LIN {X 0,Y 319.596,Z 143.485,A -85,B 0,C 180,E1 -15098.048,E2 -15098.048} C_VEL
LIN {X 0,Y 319.687,Z 143.47,A -85,B 0,C 180,E1 -15100.962,E2 -15100.962} C_VEL
LIN {X 0,Y 319.73,Z 143.468,A -85,B 0,C 180,E1 -15105.276,E2 -15105.276} C_VEL
LIN {X 0,Y 319.758,Z 143.463,A -85,B 0,C 180,E1 -15109.873,E2 -15109.873} C_VEL
LIN {X 0,Y 319.932,Z 143.443,A -85,B 0,C 180,E1 -15112.426,E2 -15112.426} C_VEL
LIN {X 0,Y 319.746,Z 143.466,A -85,B 0,C 180,E1 -15114.956,E2 -15114.956} C_VEL
LIN {X 0,Y 319.99,Z 143.436,A -85,B 0,C 180,E1 -15117.482,E2 -15117.482} C_VEL
LIN {X 0,Y 320.149,Z 143.413,A -85,B 0,C 180,E1 -15120,E2 -15120} C_VEL
LIN {X 0,Y 319.989,Z 143.434,A -85,B 0,C 180,E1 -15122.517,E2 -15122.517} C_VEL
LIN {X 0,Y 319.953,Z 143.441,A -85,B 0,C 180,E1 -15126.305,E2 -15126.305} C_VEL
LIN {X 0,Y 319.841,Z 143.451,A -85,B 0,C 180,E1 -15128.848,E2 -15128.848} C_VEL
LIN {X 0,Y 319.68,Z 143.472,A -85,B 0,C 180,E1 -15132.7,E2 -15132.7} C_VEL
LIN {X 0,Y 319.698,Z 143.476,A -85,B 0,C 180,E1 -15135.295,E2 -15135.295} C_VEL
LIN {X 0,Y 319.673,Z 143.474,A -85,B 0,C 180,E1 -15139.255,E2 -15139.255} C_VEL
LIN {X 0,Y 319.568,Z 143.491,A -85,B 0,C 180,E1 -15143.319,E2 -15143.319} C_VEL
LIN {X 0,Y 319.633,Z 143.478,A -85,B 0,C 180,E1 -15146.088,E2 -15146.088} C_VEL
LIN {X 0,Y 319.588,Z 143.487,A -85,B 0,C 180,E1 -15148.934,E2 -15148.934} C_VEL
LIN {X 0,Y 319.53,Z 143.493,A -85,B 0,C 180,E1 -15151.862,E2 -15151.862} C_VEL
LIN {X 0,Y 319.577,Z 143.485,A -85,B 0,C 180,E1 -15155.543,E2 -15155.543} C_VEL
LIN {X 0,Y 319.555,Z 143.491,A -85,B 0,C 180,E1 -15158.01,E2 -15158.01} C_VEL
LIN {X 0,Y 319.523,Z 143.488,A -85,B 0,C 180,E1 -15161.597,E2 -15161.597} C_VEL
LIN {X 0,Y 319.486,Z 143.494,A -85,B 0,C 180,E1 -15165.257,E2 -15165.257} C_VEL
LIN {X 0,Y 319.526,Z 143.494,A -85,B 0,C 180,E1 -15168.712,E2 -15168.712} C_VEL
LIN {X 0,Y 319.553,Z 143.489,A -85,B 0,C 180,E1 -15172.35,E2 -15172.35} C_VEL
LIN {X 0,Y 319.559,Z 143.49,A -85,B 0,C 180,E1 -15175.124,E2 -15175.124} C_VEL
LIN {X 0,Y 319.569,Z 143.49,A -85,B 0,C 180,E1 -15179.058,E2 -15179.058} C_VEL
LIN {X 0,Y 319.702,Z 143.582,A -85,B 0,C 180,E1 -15182.596,E2 -15182.596} C_VEL
LIN {X 0,Y 321.213,Z 151.646,A -85,B 0,C 180,E1 -15185.436,E2 -15185.436} C_VEL
LIN {X 0,Y 321.936,Z 156.902,A -85,B 0,C 180,E1 -15187.202,E2 -15187.202} C_VEL
LIN {X 0,Y 320.97,Z 166.795,A -85,B 0,C 180,E1 -15190.25,E2 -15190.25} C_VEL
LIN {X 0,Y 321.774,Z 171.894,A -85,B 0,C 180,E1 -15190.48,E2 -15190.48} C_VEL
LIN {X 0,Y 325.641,Z 196.853,A -85,B 0,C 180,E1 -15191.289,E2 -15191.289} C_VEL
LIN {X 0,Y 325.841,Z 203.062,A -85,B 0,C 180,E1 -15191.442,E2 -15191.442} C_VEL
LIN {X 0,Y 325.186,Z 243.218,A -85,B 0,C 180,E1 -15192.351,E2 -15192.351} C_VEL
LIN {X 0,Y 324.747,Z 252.267,A -85,B 0,C 180,E1 -15192.689,E2 -15192.689} C_VEL
LIN {X 0,Y 324.141,Z 261.891,A -85,B 0,C 180,E1 -15193.224,E2 -15193.224} C_VEL
LIN {X 0,Y 323.392,Z 271.027,A -85,B 0,C 180,E1 -15193.914,E2 -15193.914} C_VEL
LIN {X 0,Y 322.429,Z 281.805,A -85,B 0,C 180,E1 -15194.999,E2 -15194.999} C_VEL
LIN {X 0,Y 321.43,Z 290.08,A -85,B 0,C 180,E1 -15196.084,E2 -15196.084} C_VEL
LIN {X 0,Y 320.528,Z 297.765,A -85,B 0,C 180,E1 -15197.335,E2 -15197.335} C_VEL
LIN {X 0,Y 319.789,Z 304.092,A -85,B 0,C 180,E1 -15198.592,E2 -15198.592} C_VEL
LIN {X 0,Y 319.189,Z 309.35,A -85,B 0,C 180,E1 -15199.855,E2 -15199.855} C_VEL
LIN {X 0,Y 318.696,Z 313.734,A -85,B 0,C 180,E1 -15201.12,E2 -15201.12} C_VEL
LIN {X 0,Y 318.206,Z 318.906,A -85,B 0,C 180,E1 -15203.023,E2 -15203.023} C_VEL
LIN {X 0,Y 317.889,Z 322.703,A -85,B 0,C 180,E1 -15204.927,E2 -15204.927} C_VEL
LIN {X 0,Y 317.831,Z 324.448,A -85,B 0,C 180,E1 -15206.197,E2 -15206.197} C_VEL
LIN {X 0,Y 317.746,Z 325.696,A -85,B 0,C 180,E1 -15207.465,E2 -15207.465} C_VEL
LIN {X 0,Y 317.695,Z 326.471,A -85,B 0,C 180,E1 -15208.733,E2 -15208.733} C_VEL
LIN {X 0,Y 317.717,Z 326.765,A -85,B 0,C 180,E1 -15210,E2 -15210} C_VEL
LIN {X 0,Y 317.695,Z 326.466,A -85,B 0,C 180,E1 -15211.268,E2 -15211.268} C_VEL
LIN {X 0,Y 317.746,Z 325.679,A -85,B 0,C 180,E1 -15212.536,E2 -15212.536} C_VEL
LIN {X 0,Y 317.831,Z 324.419,A -85,B 0,C 180,E1 -15213.804,E2 -15213.804} C_VEL
LIN {X 0,Y 317.886,Z 322.663,A -85,B 0,C 180,E1 -15215.074,E2 -15215.074} C_VEL
LIN {X 0,Y 318.204,Z 318.854,A -85,B 0,C 180,E1 -15216.978,E2 -15216.978} C_VEL
LIN {X 0,Y 318.625,Z 313.665,A -85,B 0,C 180,E1 -15218.882,E2 -15218.882} C_VEL
LIN {X 0,Y 319.453,Z 306.829,A -85,B 0,C 180,E1 -15220.778,E2 -15220.778} C_VEL
LIN {X 0,Y 320.323,Z 299.357,A -85,B 0,C 180,E1 -15222.352,E2 -15222.352} C_VEL
LIN {X 0,Y 321.234,Z 291.99,A -85,B 0,C 180,E1 -15223.603,E2 -15223.603} C_VEL
LIN {X 0,Y 322.109,Z 284.099,A -85,B 0,C 180,E1 -15224.693,E2 -15224.693} C_VEL
LIN {X 0,Y 322.956,Z 275.758,A -85,B 0,C 180,E1 -15225.623,E2 -15225.623} C_VEL
LIN {X 0,Y 323.876,Z 265.096,A -85,B 0,C 180,E1 -15226.548,E2 -15226.548} C_VEL
LIN {X 0,Y 324.637,Z 253.466,A -85,B 0,C 180,E1 -15227.237,E2 -15227.237} C_VEL
LIN {X 0,Y 325.161,Z 243.694,A -85,B 0,C 180,E1 -15227.614,E2 -15227.614} C_VEL
LIN {X 0,Y 325.684,Z 197.491,A -85,B 0,C 180,E1 -15228.671,E2 -15228.671} C_VEL
LIN {X 0,Y 322.039,Z 173.379,A -85,B 0,C 180,E1 -15229.446,E2 -15229.446} C_VEL
LIN {X 0,Y 320.97,Z 166.868,A -85,B 0,C 180,E1 -15229.716,E2 -15229.716} C_VEL
LIN {X 0,Y 321.896,Z 157.872,A -85,B 0,C 180,E1 -15232.463,E2 -15232.463} C_VEL
LIN {X 0,Y 321.503,Z 153.471,A -85,B 0,C 180,E1 -15233.919,E2 -15233.919} C_VEL
LIN {X 0,Y 319.722,Z 143.707,A -85,B 0,C 180,E1 -15237.314,E2 -15237.314} C_VEL
LIN {X 0,Y 319.59,Z 143.475,A -85,B 0,C 180,E1 -15238.934,E2 -15238.934} C_VEL
LIN {X 0,Y 319.533,Z 143.496,A -85,B 0,C 180,E1 -15241.862,E2 -15241.862} C_VEL
LIN {X 0,Y 319.58,Z 143.488,A -85,B 0,C 180,E1 -15245.543,E2 -15245.543} C_VEL
LIN {X 0,Y 319.557,Z 143.486,A -85,B 0,C 180,E1 -15248.01,E2 -15248.01} C_VEL
LIN {X 0,Y 319.526,Z 143.496,A -85,B 0,C 180,E1 -15251.597,E2 -15251.597} C_VEL
LIN {X 0,Y 319.488,Z 143.494,A -85,B 0,C 180,E1 -15255.257,E2 -15255.257} C_VEL
LIN {X 0,Y 319.528,Z 143.488,A -85,B 0,C 180,E1 -15258.712,E2 -15258.712} C_VEL
LIN {X 0,Y 319.562,Z 143.489,A -85,B 0,C 180,E1 -15262.348,E2 -15262.348} C_VEL
LIN {X 0,Y 319.561,Z 143.489,A -85,B 0,C 180,E1 -15265.124,E2 -15265.124} C_VEL
LIN {X 0,Y 319.571,Z 143.492,A -85,B 0,C 180,E1 -15269.058,E2 -15269.058} C_VEL
LIN {X 0,Y 319.609,Z 143.479,A -85,B 0,C 180,E1 -15272.498,E2 -15272.498} C_VEL
LIN {X 0,Y 319.606,Z 143.486,A -85,B 0,C 180,E1 -15275.304,E2 -15275.304} C_VEL
LIN {X 0,Y 319.599,Z 143.483,A -85,B 0,C 180,E1 -15278.048,E2 -15278.048} C_VEL
LIN {X 0,Y 319.69,Z 143.472,A -85,B 0,C 180,E1 -15280.962,E2 -15280.962} C_VEL
LIN {X 0,Y 319.732,Z 143.468,A -85,B 0,C 180,E1 -15285.276,E2 -15285.276} C_VEL
LIN {X 0,Y 319.754,Z 143.458,A -85,B 0,C 180,E1 -15289.873,E2 -15289.873} C_VEL
LIN {X 0,Y 319.914,Z 143.449,A -85,B 0,C 180,E1 -15292.426,E2 -15292.426} C_VEL
LIN {X 0,Y 319.746,Z 143.466,A -85,B 0,C 180,E1 -15294.956,E2 -15294.956} C_VEL
LIN {X 0,Y 319.991,Z 143.433,A -85,B 0,C 180,E1 -15297.483,E2 -15297.483} C_VEL
LIN {X 0,Y 320.133,Z 143.415,A -85,B 0,C 180,E1 -15300,E2 -15300} C_VEL
LIN {X 0,Y 319.991,Z 143.436,A -85,B 0,C 180,E1 -15302.518,E2 -15302.518} C_VEL
LIN {X 0,Y 319.934,Z 143.44,A -85,B 0,C 180,E1 -15306.638,E2 -15306.638} C_VEL
LIN {X 0,Y 319.762,Z 143.463,A -85,B 0,C 180,E1 -15310.127,E2 -15310.127} C_VEL
LIN {X 0,Y 319.733,Z 143.467,A -85,B 0,C 180,E1 -15314.724,E2 -15314.724} C_VEL
LIN {X 0,Y 319.691,Z 143.469,A -85,B 0,C 180,E1 -15319.038,E2 -15319.038} C_VEL
LIN {X 0,Y 319.572,Z 143.491,A -85,B 0,C 180,E1 -15323.319,E2 -15323.319} C_VEL
LIN {X 0,Y 319.62,Z 143.477,A -85,B 0,C 180,E1 -15326.089,E2 -15326.089} C_VEL
LIN {X 0,Y 319.591,Z 143.488,A -85,B 0,C 180,E1 -15328.934,E2 -15328.934} C_VEL
LIN {X 0,Y 319.534,Z 143.492,A -85,B 0,C 180,E1 -15331.862,E2 -15331.862} C_VEL
LIN {X 0,Y 319.581,Z 143.486,A -85,B 0,C 180,E1 -15335.543,E2 -15335.543} C_VEL
LIN {X 0,Y 319.559,Z 143.49,A -85,B 0,C 180,E1 -15338.01,E2 -15338.01} C_VEL
LIN {X 0,Y 319.527,Z 143.493,A -85,B 0,C 180,E1 -15341.597,E2 -15341.597} C_VEL
LIN {X 0,Y 319.49,Z 143.495,A -85,B 0,C 180,E1 -15345.257,E2 -15345.257} C_VEL
LIN {X 0,Y 319.53,Z 143.49,A -85,B 0,C 180,E1 -15348.712,E2 -15348.712} C_VEL
LIN {X 0,Y 319.579,Z 143.489,A -85,B 0,C 180,E1 -15352.344,E2 -15352.344} C_VEL
LIN {X 0,Y 319.562,Z 143.48,A -85,B 0,C 180,E1 -15355.123,E2 -15355.123} C_VEL
LIN {X 0,Y 319.572,Z 143.488,A -85,B 0,C 180,E1 -15359.058,E2 -15359.058} C_VEL
LIN {X 0,Y 319.61,Z 143.483,A -85,B 0,C 180,E1 -15362.498,E2 -15362.498} C_VEL
LIN {X 0,Y 319.635,Z 143.653,A -85,B 0,C 180,E1 -15365.955,E2 -15365.955} C_VEL
LIN {X 0,Y 321.074,Z 151.506,A -85,B 0,C 180,E1 -15368.828,E2 -15368.828} C_VEL
LIN {X 0,Y 321.228,Z 156.146,A -85,B 0,C 180,E1 -15370.342,E2 -15370.342} C_VEL
LIN {X 0,Y 321.834,Z 159.261,A -85,B 0,C 180,E1 -15370.514,E2 -15370.514} C_VEL
LIN {X 0,Y 326.078,Z 182.285,A -85,B 0,C 180,E1 -15371.305,E2 -15371.305} C_VEL
LIN {X 0,Y 325.231,Z 232.335,A -85,B 0,C 180,E1 -15372.431,E2 -15372.431} C_VEL
LIN {X 0,Y 324.852,Z 242.15,A -85,B 0,C 180,E1 -15372.815,E2 -15372.815} C_VEL
LIN {X 0,Y 324.282,Z 253.252,A -85,B 0,C 180,E1 -15373.474,E2 -15373.474} C_VEL
LIN {X 0,Y 323.393,Z 264.079,A -85,B 0,C 180,E1 -15374.399,E2 -15374.399} C_VEL
LIN {X 0,Y 322.546,Z 272.474,A -85,B 0,C 180,E1 -15375.327,E2 -15375.327} C_VEL
LIN {X 0,Y 321.773,Z 280.397,A -85,B 0,C 180,E1 -15376.42,E2 -15376.42} C_VEL
LIN {X 0,Y 321.069,Z 286.089,A -85,B 0,C 180,E1 -15377.356,E2 -15377.356} C_VEL
LIN {X 0,Y 320.328,Z 292.441,A -85,B 0,C 180,E1 -15378.611,E2 -15378.611} C_VEL
LIN {X 0,Y 319.592,Z 297.723,A -85,B 0,C 180,E1 -15379.867,E2 -15379.867} C_VEL
LIN {X 0,Y 319.125,Z 302.13,A -85,B 0,C 180,E1 -15381.132,E2 -15381.132} C_VEL
LIN {X 0,Y 318.731,Z 305.8,A -85,B 0,C 180,E1 -15382.397,E2 -15382.397} C_VEL
LIN {X 0,Y 318.383,Z 308.798,A -85,B 0,C 180,E1 -15383.663,E2 -15383.663} C_VEL
LIN {X 0,Y 318.189,Z 311.118,A -85,B 0,C 180,E1 -15384.931,E2 -15384.931} C_VEL
LIN {X 0,Y 317.988,Z 312.884,A -85,B 0,C 180,E1 -15386.198,E2 -15386.198} C_VEL
LIN {X 0,Y 317.81,Z 314.158,A -85,B 0,C 180,E1 -15387.465,E2 -15387.465} C_VEL
LIN {X 0,Y 317.725,Z 314.961,A -85,B 0,C 180,E1 -15388.732,E2 -15388.732} C_VEL
LIN {X 0,Y 317.721,Z 315.267,A -85,B 0,C 180,E1 -15390,E2 -15390} C_VEL
LIN {X 0,Y 317.725,Z 314.99,A -85,B 0,C 180,E1 -15391.267,E2 -15391.267} C_VEL
LIN {X 0,Y 317.808,Z 314.243,A -85,B 0,C 180,E1 -15392.535,E2 -15392.535} C_VEL
LIN {X 0,Y 317.984,Z 313.027,A -85,B 0,C 180,E1 -15393.801,E2 -15393.801} C_VEL
LIN {X 0,Y 318.265,Z 310.175,A -85,B 0,C 180,E1 -15395.703,E2 -15395.703} C_VEL
LIN {X 0,Y 318.578,Z 307.161,A -85,B 0,C 180,E1 -15397.144,E2 -15397.144} C_VEL
LIN {X 0,Y 319.063,Z 302.468,A -85,B 0,C 180,E1 -15398.869,E2 -15398.869} C_VEL
LIN {X 0,Y 319.729,Z 296.969,A -85,B 0,C 180,E1 -15400.448,E2 -15400.448} C_VEL
LIN {X 0,Y 320.595,Z 290.059,A -85,B 0,C 180,E1 -15402.02,E2 -15402.02} C_VEL
LIN {X 0,Y 321.555,Z 282.123,A -85,B 0,C 180,E1 -15403.428,E2 -15403.428} C_VEL
LIN {X 0,Y 322.403,Z 274.555,A -85,B 0,C 180,E1 -15404.518,E2 -15404.518} C_VEL
LIN {X 0,Y 323.255,Z 266.621,A -85,B 0,C 180,E1 -15405.446,E2 -15405.446} C_VEL
LIN {X 0,Y 323.921,Z 258.426,A -85,B 0,C 180,E1 -15406.221,E2 -15406.221} C_VEL
LIN {X 0,Y 324.56,Z 250.118,A -85,B 0,C 180,E1 -15406.835,E2 -15406.835} C_VEL
LIN {X 0,Y 325.022,Z 241.136,A -85,B 0,C 180,E1 -15407.337,E2 -15407.337} C_VEL
LIN {X 0,Y 325.384,Z 231.483,A -85,B 0,C 180,E1 -15407.7,E2 -15407.7} C_VEL
LIN {X 0,Y 326.088,Z 182.324,A -85,B 0,C 180,E1 -15408.806,E2 -15408.806} C_VEL
LIN {X 0,Y 321.573,Z 158.002,A -85,B 0,C 180,E1 -15409.646,E2 -15409.646} C_VEL
LIN {X 0,Y 321.227,Z 156.132,A -85,B 0,C 180,E1 -15409.774,E2 -15409.774} C_VEL
LIN {X 0,Y 321.084,Z 151.844,A -85,B 0,C 180,E1 -15411.171,E2 -15411.171} C_VEL
LIN {X 0,Y 319.679,Z 143.603,A -85,B 0,C 180,E1 -15414.192,E2 -15414.192} C_VEL
LIN {X 0,Y 319.609,Z 143.482,A -85,B 0,C 180,E1 -15417.501,E2 -15417.501} C_VEL
LIN {X 0,Y 319.57,Z 143.488,A -85,B 0,C 180,E1 -15420.942,E2 -15420.942} C_VEL
LIN {X 0,Y 319.56,Z 143.481,A -85,B 0,C 180,E1 -15424.876,E2 -15424.876} C_VEL
LIN {X 0,Y 319.57,Z 143.492,A -85,B 0,C 180,E1 -15428.037,E2 -15428.037} C_VEL
LIN {X 0,Y 319.525,Z 143.489,A -85,B 0,C 180,E1 -15431.597,E2 -15431.597} C_VEL
LIN {X 0,Y 319.515,Z 143.485,A -85,B 0,C 180,E1 -15433.527,E2 -15433.527} C_VEL
LIN {X 0,Y 318.79,Z 143.583,A -85,B 0,C 180,E1 -15434.578,E2 -15434.578} C_VEL
LIN {X 0,Y 315.91,Z 143.945,A -85,B 0,C 180,E1 -15436.289,E2 -15436.289} C_VEL
LIN {X 0,Y 313.527,Z 144.245,A -85,B 0,C 180,E1 -15437.676,E2 -15437.676} C_VEL
LIN {X 0,Y 312.541,Z 144.364,A -85,B 0,C 180,E1 -15438.75,E2 -15438.75} C_VEL
LIN {X 0,Y 312.478,Z 144.373,A -85,B 0,C 180,E1 -15439.113,E2 -15439.113} C_VEL
LIN {X 0,Y 312.524,Z 144.366,A -85,B 0,C 180,E1 -15442.615,E2 -15442.615} C_VEL
LIN {X 0,Y 312.518,Z 144.361,A -85,B 0,C 180,E1 -15446.311,E2 -15446.311} C_VEL
LIN {X 0,Y 312.544,Z 144.363,A -85,B 0,C 180,E1 -15450.35,E2 -15450.35} C_VEL
LIN {X 0,Y 312.596,Z 144.351,A -85,B 0,C 180,E1 -15454.066,E2 -15454.066} C_VEL
LIN {X 0,Y 312.586,Z 144.358,A -85,B 0,C 180,E1 -15457.529,E2 -15457.529} C_VEL
LIN {X 0,Y 312.637,Z 144.344,A -85,B 0,C 180,E1 -15461.656,E2 -15461.656} C_VEL
LIN {X 0,Y 312.693,Z 144.344,A -85,B 0,C 180,E1 -15465.686,E2 -15465.686} C_VEL
LIN {X 0,Y 312.703,Z 144.34,A -85,B 0,C 180,E1 -15469.642,E2 -15469.642} C_VEL
LIN {X 0,Y 312.87,Z 144.32,A -85,B 0,C 180,E1 -15472.254,E2 -15472.254} C_VEL
LIN {X 0,Y 312.716,Z 144.342,A -85,B 0,C 180,E1 -15474.842,E2 -15474.842} C_VEL
LIN {X 0,Y 312.989,Z 144.304,A -85,B 0,C 180,E1 -15478.713,E2 -15478.713} C_VEL
LIN {X 0,Y 312.989,Z 144.3,A -85,B 0,C 180,E1 -15481.287,E2 -15481.287} C_VEL
LIN {X 0,Y 312.718,Z 144.342,A -85,B 0,C 180,E1 -15485.157,E2 -15485.157} C_VEL
LIN {X 0,Y 312.871,Z 144.324,A -85,B 0,C 180,E1 -15487.746,E2 -15487.746} C_VEL
LIN {X 0,Y 312.667,Z 144.347,A -85,B 0,C 180,E1 -15491.671,E2 -15491.671} C_VEL
LIN {X 0,Y 312.698,Z 144.345,A -85,B 0,C 180,E1 -15494.888,E2 -15494.888} C_VEL
LIN {X 0,Y 312.628,Z 144.35,A -85,B 0,C 180,E1 -15499.236,E2 -15499.236} C_VEL
LIN {X 0,Y 312.544,Z 144.365,A -85,B 0,C 180,E1 -15502.789,E2 -15502.789} C_VEL
LIN {X 0,Y 312.581,Z 144.359,A -85,B 0,C 180,E1 -15506.723,E2 -15506.723} C_VEL
LIN {X 0,Y 312.543,Z 144.362,A -85,B 0,C 180,E1 -15509.65,E2 -15509.65} C_VEL
LIN {X 0,Y 312.517,Z 144.364,A -85,B 0,C 180,E1 -15513.689,E2 -15513.689} C_VEL
LIN {X 0,Y 312.523,Z 144.366,A -85,B 0,C 180,E1 -15517.385,E2 -15517.385} C_VEL
LIN {X 0,Y 312.488,Z 144.367,A -85,B 0,C 180,E1 -15520.709,E2 -15520.709} C_VEL
LIN {X 0,Y 312.449,Z 144.363,A -85,B 0,C 180,E1 -15524.21,E2 -15524.21} C_VEL
LIN {X 0,Y 312.482,Z 144.374,A -85,B 0,C 180,E1 -15527.919,E2 -15527.919} C_VEL
LIN {X 0,Y 312.497,Z 144.363,A -85,B 0,C 180,E1 -15530.971,E2 -15530.971} C_VEL
LIN {X 0,Y 312.53,Z 144.368,A -85,B 0,C 180,E1 -15534.221,E2 -15534.221} C_VEL
LIN {X 0,Y 312.504,Z 144.365,A -85,B 0,C 180,E1 -15537.334,E2 -15537.334} C_VEL
LIN {X 0,Y 312.55,Z 144.344,A -85,B 0,C 180,E1 -15541.277,E2 -15541.277} C_VEL
LIN {X 0,Y 312.634,Z 144.484,A -85,B 0,C 180,E1 -15542.287,E2 -15542.287} C_VEL
LIN {X 0,Y 314.194,Z 152.563,A -85,B 0,C 180,E1 -15545.204,E2 -15545.204} C_VEL
LIN {X 0,Y 314.96,Z 157.818,A -85,B 0,C 180,E1 -15547.015,E2 -15547.015} C_VEL
LIN {X 0,Y 314.083,Z 166.45,A -85,B 0,C 180,E1 -15549.756,E2 -15549.756} C_VEL
LIN {X 0,Y 314.392,Z 168.734,A -85,B 0,C 180,E1 -15549.93,E2 -15549.93} C_VEL
LIN {X 0,Y 318.64,Z 195.359,A -85,B 0,C 180,E1 -15550.83,E2 -15550.83} C_VEL
LIN {X 0,Y 319.138,Z 202.091,A -85,B 0,C 180,E1 -15551.018,E2 -15551.018} C_VEL
LIN {X 0,Y 318.413,Z 243.216,A -85,B 0,C 180,E1 -15551.966,E2 -15551.966} C_VEL
LIN {X 0,Y 317.919,Z 252.979,A -85,B 0,C 180,E1 -15552.346,E2 -15552.346} C_VEL
LIN {X 0,Y 317.288,Z 262.98,A -85,B 0,C 180,E1 -15552.933,E2 -15552.933} C_VEL
LIN {X 0,Y 316.28,Z 274.341,A -85,B 0,C 180,E1 -15553.874,E2 -15553.874} C_VEL
LIN {X 0,Y 315.41,Z 282.912,A -85,B 0,C 180,E1 -15554.823,E2 -15554.823} C_VEL
LIN {X 0,Y 314.397,Z 290.976,A -85,B 0,C 180,E1 -15555.931,E2 -15555.931} C_VEL
LIN {X 0,Y 313.588,Z 297.639,A -85,B 0,C 180,E1 -15557.049,E2 -15557.049} C_VEL
LIN {X 0,Y 312.824,Z 303.966,A -85,B 0,C 180,E1 -15558.335,E2 -15558.335} C_VEL
LIN {X 0,Y 312.197,Z 309.223,A -85,B 0,C 180,E1 -15559.625,E2 -15559.625} C_VEL
LIN {X 0,Y 311.661,Z 313.607,A -85,B 0,C 180,E1 -15560.918,E2 -15560.918} C_VEL
LIN {X 0,Y 311.133,Z 318.778,A -85,B 0,C 180,E1 -15562.864,E2 -15562.864} C_VEL
LIN {X 0,Y 310.807,Z 322.575,A -85,B 0,C 180,E1 -15564.811,E2 -15564.811} C_VEL
LIN {X 0,Y 310.745,Z 324.32,A -85,B 0,C 180,E1 -15566.11,E2 -15566.11} C_VEL
LIN {X 0,Y 310.672,Z 325.568,A -85,B 0,C 180,E1 -15567.407,E2 -15567.407} C_VEL
LIN {X 0,Y 310.612,Z 326.343,A -85,B 0,C 180,E1 -15568.704,E2 -15568.704} C_VEL
LIN {X 0,Y 310.629,Z 326.637,A -85,B 0,C 180,E1 -15570,E2 -15570} C_VEL
LIN {X 0,Y 310.612,Z 326.338,A -85,B 0,C 180,E1 -15571.297,E2 -15571.297} C_VEL
LIN {X 0,Y 310.672,Z 325.551,A -85,B 0,C 180,E1 -15572.593,E2 -15572.593} C_VEL
LIN {X 0,Y 310.745,Z 324.29,A -85,B 0,C 180,E1 -15573.891,E2 -15573.891} C_VEL
LIN {X 0,Y 310.889,Z 321.236,A -85,B 0,C 180,E1 -15575.919,E2 -15575.919} C_VEL
LIN {X 0,Y 311.258,Z 317.201,A -85,B 0,C 180,E1 -15577.786,E2 -15577.786} C_VEL
LIN {X 0,Y 311.899,Z 311.486,A -85,B 0,C 180,E1 -15579.73,E2 -15579.73} C_VEL
LIN {X 0,Y 312.638,Z 305.282,A -85,B 0,C 180,E1 -15581.344,E2 -15581.344} C_VEL
LIN {X 0,Y 313.374,Z 299.226,A -85,B 0,C 180,E1 -15582.631,E2 -15582.631} C_VEL
LIN {X 0,Y 314.34,Z 291.859,A -85,B 0,C 180,E1 -15583.907,E2 -15583.907} C_VEL
LIN {X 0,Y 315.239,Z 283.967,A -85,B 0,C 180,E1 -15585.021,E2 -15585.021} C_VEL
LIN {X 0,Y 316.137,Z 275.626,A -85,B 0,C 180,E1 -15585.969,E2 -15585.969} C_VEL
LIN {X 0,Y 317.071,Z 264.961,A -85,B 0,C 180,E1 -15586.913,E2 -15586.913} C_VEL
LIN {X 0,Y 317.875,Z 253.328,A -85,B 0,C 180,E1 -15587.615,E2 -15587.615} C_VEL
LIN {X 0,Y 318.411,Z 243.551,A -85,B 0,C 180,E1 -15588,E2 -15588} C_VEL
LIN {X 0,Y 318.975,Z 198.24,A -85,B 0,C 180,E1 -15589.058,E2 -15589.058} C_VEL
LIN {X 0,Y 315.446,Z 174.945,A -85,B 0,C 180,E1 -15589.829,E2 -15589.829} C_VEL
LIN {X 0,Y 314.079,Z 167.022,A -85,B 0,C 180,E1 -15590.135,E2 -15590.135} C_VEL
LIN {X 0,Y 314.097,Z 165.965,A -85,B 0,C 180,E1 -15590.352,E2 -15590.352} C_VEL
LIN {X 0,Y 314.923,Z 158.785,A -85,B 0,C 180,E1 -15592.642,E2 -15592.642} C_VEL
LIN {X 0,Y 314.331,Z 153.532,A -85,B 0,C 180,E1 -15594.434,E2 -15594.434} C_VEL
LIN {X 0,Y 312.636,Z 144.451,A -85,B 0,C 180,E1 -15597.714,E2 -15597.714} C_VEL
LIN {X 0,Y 312.518,Z 144.368,A -85,B 0,C 180,E1 -15601.289,E2 -15601.289} C_VEL
LIN {X 0,Y 312.507,Z 144.369,A -85,B 0,C 180,E1 -15604.21,E2 -15604.21} C_VEL
LIN {X 0,Y 312.526,Z 144.363,A -85,B 0,C 180,E1 -15607.385,E2 -15607.385} C_VEL
LIN {X 0,Y 312.49,Z 144.37,A -85,B 0,C 180,E1 -15610.709,E2 -15610.709} C_VEL
LIN {X 0,Y 312.452,Z 144.37,A -85,B 0,C 180,E1 -15614.21,E2 -15614.21} C_VEL
LIN {X 0,Y 312.484,Z 144.364,A -85,B 0,C 180,E1 -15617.919,E2 -15617.919} C_VEL
LIN {X 0,Y 312.506,Z 144.37,A -85,B 0,C 180,E1 -15621.918,E2 -15621.918} C_VEL
LIN {X 0,Y 312.532,Z 144.362,A -85,B 0,C 180,E1 -15624.221,E2 -15624.221} C_VEL
LIN {X 0,Y 312.505,Z 144.372,A -85,B 0,C 180,E1 -15627.334,E2 -15627.334} C_VEL
LIN {X 0,Y 312.553,Z 144.36,A -85,B 0,C 180,E1 -15631.276,E2 -15631.276} C_VEL
LIN {X 0,Y 312.587,Z 144.359,A -85,B 0,C 180,E1 -15634.711,E2 -15634.711} C_VEL
LIN {X 0,Y 312.589,Z 144.357,A -85,B 0,C 180,E1 -15637.529,E2 -15637.529} C_VEL
LIN {X 0,Y 312.64,Z 144.348,A -85,B 0,C 180,E1 -15641.657,E2 -15641.657} C_VEL
LIN {X 0,Y 312.695,Z 144.344,A -85,B 0,C 180,E1 -15645.686,E2 -15645.686} C_VEL
LIN {X 0,Y 312.7,Z 144.335,A -85,B 0,C 180,E1 -15649.642,E2 -15649.642} C_VEL
LIN {X 0,Y 312.855,Z 144.326,A -85,B 0,C 180,E1 -15652.254,E2 -15652.254} C_VEL
LIN {X 0,Y 312.716,Z 144.342,A -85,B 0,C 180,E1 -15654.843,E2 -15654.843} C_VEL
LIN {X 0,Y 312.99,Z 144.3,A -85,B 0,C 180,E1 -15658.713,E2 -15658.713} C_VEL
LIN {X 0,Y 312.99,Z 144.304,A -85,B 0,C 180,E1 -15661.287,E2 -15661.287} C_VEL
LIN {X 0,Y 312.718,Z 144.342,A -85,B 0,C 180,E1 -15665.158,E2 -15665.158} C_VEL
LIN {X 0,Y 312.874,Z 144.32,A -85,B 0,C 180,E1 -15667.746,E2 -15667.746} C_VEL
LIN {X 0,Y 312.674,Z 144.349,A -85,B 0,C 180,E1 -15671.671,E2 -15671.671} C_VEL
LIN {X 0,Y 312.702,Z 144.344,A -85,B 0,C 180,E1 -15674.888,E2 -15674.888} C_VEL
LIN {X 0,Y 312.632,Z 144.349,A -85,B 0,C 180,E1 -15679.237,E2 -15679.237} C_VEL
LIN {X 0,Y 312.548,Z 144.364,A -85,B 0,C 180,E1 -15682.789,E2 -15682.789} C_VEL
LIN {X 0,Y 312.599,Z 144.351,A -85,B 0,C 180,E1 -15685.933,E2 -15685.933} C_VEL
LIN {X 0,Y 312.547,Z 144.363,A -85,B 0,C 180,E1 -15689.65,E2 -15689.65} C_VEL
LIN {X 0,Y 312.521,Z 144.361,A -85,B 0,C 180,E1 -15693.689,E2 -15693.689} C_VEL
LIN {X 0,Y 312.527,Z 144.366,A -85,B 0,C 180,E1 -15697.385,E2 -15697.385} C_VEL
LIN {X 0,Y 312.491,Z 144.372,A -85,B 0,C 180,E1 -15700.709,E2 -15700.709} C_VEL
LIN {X 0,Y 312.453,Z 144.378,A -85,B 0,C 180,E1 -15704.21,E2 -15704.21} C_VEL
LIN {X 0,Y 312.486,Z 144.36,A -85,B 0,C 180,E1 -15707.919,E2 -15707.919} C_VEL
LIN {X 0,Y 312.537,Z 144.368,A -85,B 0,C 180,E1 -15711.91,E2 -15711.91} C_VEL
LIN {X 0,Y 312.508,Z 144.361,A -85,B 0,C 180,E1 -15715.79,E2 -15715.79} C_VEL
LIN {X 0,Y 312.526,Z 144.365,A -85,B 0,C 180,E1 -15718.854,E2 -15718.854} C_VEL
LIN {X 0,Y 312.576,Z 144.363,A -85,B 0,C 180,E1 -15721.825,E2 -15721.825} C_VEL
LIN {X 0,Y 312.606,Z 144.466,A -85,B 0,C 180,E1 -15725.6,E2 -15725.6} C_VEL
LIN {X 0,Y 313.942,Z 151.636,A -85,B 0,C 180,E1 -15728.323,E2 -15728.323} C_VEL
LIN {X 0,Y 314.28,Z 156.159,A -85,B 0,C 180,E1 -15729.87,E2 -15729.87} C_VEL
LIN {X 0,Y 314.743,Z 158.525,A -85,B 0,C 180,E1 -15730.035,E2 -15730.035} C_VEL
LIN {X 0,Y 319.257,Z 182.327,A -85,B 0,C 180,E1 -15730.888,E2 -15730.888} C_VEL
LIN {X 0,Y 318.483,Z 232.481,A -85,B 0,C 180,E1 -15732.046,E2 -15732.046} C_VEL
LIN {X 0,Y 318.097,Z 242.289,A -85,B 0,C 180,E1 -15732.439,E2 -15732.439} C_VEL
LIN {X 0,Y 317.5,Z 253.388,A -85,B 0,C 180,E1 -15733.11,E2 -15733.11} C_VEL
LIN {X 0,Y 316.553,Z 264.212,A -85,B 0,C 180,E1 -15734.053,E2 -15734.053} C_VEL
LIN {X 0,Y 315.701,Z 272.606,A -85,B 0,C 180,E1 -15735.001,E2 -15735.001} C_VEL
LIN {X 0,Y 314.883,Z 280.529,A -85,B 0,C 180,E1 -15736.117,E2 -15736.117} C_VEL
LIN {X 0,Y 314.155,Z 286.22,A -85,B 0,C 180,E1 -15737.073,E2 -15737.073} C_VEL
LIN {X 0,Y 313.379,Z 292.572,A -85,B 0,C 180,E1 -15738.355,E2 -15738.355} C_VEL
LIN {X 0,Y 312.599,Z 297.854,A -85,B 0,C 180,E1 -15739.638,E2 -15739.638} C_VEL
LIN {X 0,Y 312.089,Z 302.261,A -85,B 0,C 180,E1 -15740.93,E2 -15740.93} C_VEL
LIN {X 0,Y 311.688,Z 305.93,A -85,B 0,C 180,E1 -15742.224,E2 -15742.224} C_VEL
LIN {X 0,Y 311.255,Z 309.55,A -85,B 0,C 180,E1 -15743.855,E2 -15743.855} C_VEL
LIN {X 0,Y 311.124,Z 311.248,A -85,B 0,C 180,E1 -15744.816,E2 -15744.816} C_VEL
LIN {X 0,Y 310.926,Z 313.013,A -85,B 0,C 180,E1 -15746.111,E2 -15746.111} C_VEL
LIN {X 0,Y 310.736,Z 314.286,A -85,B 0,C 180,E1 -15747.407,E2 -15747.407} C_VEL
LIN {X 0,Y 310.641,Z 315.09,A -85,B 0,C 180,E1 -15748.703,E2 -15748.703} C_VEL
LIN {X 0,Y 310.634,Z 315.395,A -85,B 0,C 180,E1 -15750,E2 -15750} C_VEL
LIN {X 0,Y 310.641,Z 315.118,A -85,B 0,C 180,E1 -15751.296,E2 -15751.296} C_VEL
LIN {X 0,Y 310.735,Z 314.371,A -85,B 0,C 180,E1 -15752.592,E2 -15752.592} C_VEL
LIN {X 0,Y 310.922,Z 313.155,A -85,B 0,C 180,E1 -15753.888,E2 -15753.888} C_VEL
LIN {X 0,Y 311.111,Z 311.449,A -85,B 0,C 180,E1 -15755.184,E2 -15755.184} C_VEL
LIN {X 0,Y 311.452,Z 307.857,A -85,B 0,C 180,E1 -15757.064,E2 -15757.064} C_VEL
LIN {X 0,Y 312.034,Z 302.596,A -85,B 0,C 180,E1 -15759.071,E2 -15759.071} C_VEL
LIN {X 0,Y 312.764,Z 297.095,A -85,B 0,C 180,E1 -15760.683,E2 -15760.683} C_VEL
LIN {X 0,Y 313.662,Z 290.185,A -85,B 0,C 180,E1 -15762.29,E2 -15762.29} C_VEL
LIN {X 0,Y 314.664,Z 282.248,A -85,B 0,C 180,E1 -15763.727,E2 -15763.727} C_VEL
LIN {X 0,Y 315.543,Z 274.679,A -85,B 0,C 180,E1 -15764.841,E2 -15764.841} C_VEL
LIN {X 0,Y 316.435,Z 266.744,A -85,B 0,C 180,E1 -15765.787,E2 -15765.787} C_VEL
LIN {X 0,Y 317.126,Z 258.548,A -85,B 0,C 180,E1 -15766.578,E2 -15766.578} C_VEL
LIN {X 0,Y 317.783,Z 250.238,A -85,B 0,C 180,E1 -15767.205,E2 -15767.205} C_VEL
LIN {X 0,Y 318.276,Z 241.253,A -85,B 0,C 180,E1 -15767.716,E2 -15767.716} C_VEL
LIN {X 0,Y 318.619,Z 231.956,A -85,B 0,C 180,E1 -15768.077,E2 -15768.077} C_VEL
LIN {X 0,Y 319.393,Z 183.347,A -85,B 0,C 180,E1 -15769.194,E2 -15769.194} C_VEL
LIN {X 0,Y 314.998,Z 159.545,A -85,B 0,C 180,E1 -15770.039,E2 -15770.039} C_VEL
LIN {X 0,Y 314.286,Z 156.315,A -85,B 0,C 180,E1 -15770.221,E2 -15770.221} C_VEL
LIN {X 0,Y 313.958,Z 151.969,A -85,B 0,C 180,E1 -15771.675,E2 -15771.675} C_VEL
LIN {X 0,Y 312.622,Z 144.463,A -85,B 0,C 180,E1 -15774.531,E2 -15774.531} C_VEL
LIN {X 0,Y 312.575,Z 144.362,A -85,B 0,C 180,E1 -15778.175,E2 -15778.175} C_VEL
LIN {X 0,Y 312.518,Z 144.366,A -85,B 0,C 180,E1 -15781.289,E2 -15781.289} C_VEL
LIN {X 0,Y 312.506,Z 144.363,A -85,B 0,C 180,E1 -15784.21,E2 -15784.21} C_VEL
LIN {X 0,Y 312.534,Z 144.369,A -85,B 0,C 180,E1 -15788.089,E2 -15788.089} C_VEL
LIN {X 0,Y 312.483,Z 144.358,A -85,B 0,C 180,E1 -15792.081,E2 -15792.081} C_VEL
LIN {X 0,Y 312.457,Z 144.376,A -85,B 0,C 180,E1 -15796.035,E2 -15796.035} C_VEL
LIN {X 0,Y 312.478,Z 144.373,A -85,B 0,C 180,E1 -15799.113,E2 -15799.113} C_VEL
LIN {X 0,Y 311.849,Z 144.455,A -85,B 0,C 180,E1 -15800.188,E2 -15800.188} C_VEL
LIN {X 0,Y 308.988,Z 144.809,A -85,B 0,C 180,E1 -15801.938,E2 -15801.938} C_VEL
LIN {X 0,Y 306.552,Z 145.115,A -85,B 0,C 180,E1 -15803.357,E2 -15803.357} C_VEL
LIN {X 0,Y 305.529,Z 145.237,A -85,B 0,C 180,E1 -15804.456,E2 -15804.456} C_VEL
LIN {X 0,Y 305.459,Z 145.247,A -85,B 0,C 180,E1 -15804.828,E2 -15804.828} C_VEL
LIN {X 0,Y 305.45,Z 145.246,A -85,B 0,C 180,E1 -15808.355,E2 -15808.355} C_VEL
LIN {X 0,Y 305.519,Z 145.241,A -85,B 0,C 180,E1 -15811.114,E2 -15811.114} C_VEL
LIN {X 0,Y 305.564,Z 145.226,A -85,B 0,C 180,E1 -15814.087,E2 -15814.087} C_VEL
LIN {X 0,Y 305.5,Z 145.242,A -85,B 0,C 180,E1 -15818.403,E2 -15818.403} C_VEL
LIN {X 0,Y 305.589,Z 145.222,A -85,B 0,C 180,E1 -15821.217,E2 -15821.217} C_VEL
LIN {X 0,Y 305.648,Z 145.222,A -85,B 0,C 180,E1 -15825.349,E2 -15825.349} C_VEL
LIN {X 0,Y 305.639,Z 145.219,A -85,B 0,C 180,E1 -15829.4,E2 -15829.4} C_VEL
LIN {X 0,Y 305.811,Z 145.196,A -85,B 0,C 180,E1 -15832.074,E2 -15832.074} C_VEL
LIN {X 0,Y 305.688,Z 145.218,A -85,B 0,C 180,E1 -15834.723,E2 -15834.723} C_VEL
LIN {X 0,Y 305.956,Z 145.18,A -85,B 0,C 180,E1 -15838.684,E2 -15838.684} C_VEL
LIN {X 0,Y 305.956,Z 145.175,A -85,B 0,C 180,E1 -15841.316,E2 -15841.316} C_VEL
LIN {X 0,Y 305.853,Z 145.196,A -85,B 0,C 180,E1 -15846.597,E2 -15846.597} C_VEL
LIN {X 0,Y 305.734,Z 145.21,A -85,B 0,C 180,E1 -15849.26,E2 -15849.26} C_VEL
LIN {X 0,Y 305.587,Z 145.23,A -85,B 0,C 180,E1 -15853.296,E2 -15853.296} C_VEL
LIN {X 0,Y 305.592,Z 145.229,A -85,B 0,C 180,E1 -15856.02,E2 -15856.02} C_VEL
LIN {X 0,Y 305.575,Z 145.227,A -85,B 0,C 180,E1 -15859.445,E2 -15859.445} C_VEL
LIN {X 0,Y 305.489,Z 145.246,A -85,B 0,C 180,E1 -15863.042,E2 -15863.042} C_VEL
LIN {X 0,Y 305.552,Z 145.232,A -85,B 0,C 180,E1 -15866.23,E2 -15866.23} C_VEL
LIN {X 0,Y 305.494,Z 145.242,A -85,B 0,C 180,E1 -15869.05,E2 -15869.05} C_VEL
LIN {X 0,Y 305.463,Z 145.243,A -85,B 0,C 180,E1 -15873.517,E2 -15873.517} C_VEL
LIN {X 0,Y 305.473,Z 145.248,A -85,B 0,C 180,E1 -15876.74,E2 -15876.74} C_VEL
LIN {X 0,Y 305.452,Z 145.243,A -85,B 0,C 180,E1 -15880.6,E2 -15880.6} C_VEL
LIN {X 0,Y 305.423,Z 145.232,A -85,B 0,C 180,E1 -15883.655,E2 -15883.655} C_VEL
LIN {X 0,Y 305.453,Z 145.247,A -85,B 0,C 180,E1 -15887.414,E2 -15887.414} C_VEL
LIN {X 0,Y 305.466,Z 145.238,A -85,B 0,C 180,E1 -15891.597,E2 -15891.597} C_VEL
LIN {X 0,Y 305.461,Z 145.247,A -85,B 0,C 180,E1 -15894.887,E2 -15894.887} C_VEL
LIN {X 0,Y 305.451,Z 145.25,A -85,B 0,C 180,E1 -15898.355,E2 -15898.355} C_VEL
LIN {X 0,Y 305.584,Z 145.386,A -85,B 0,C 180,E1 -15901.964,E2 -15901.964} C_VEL
LIN {X 0,Y 307.336,Z 154.531,A -85,B 0,C 180,E1 -15905.334,E2 -15905.334} C_VEL
LIN {X 0,Y 307.976,Z 159.782,A -85,B 0,C 180,E1 -15907.174,E2 -15907.174} C_VEL
LIN {X 0,Y 307.194,Z 166.597,A -85,B 0,C 180,E1 -15909.332,E2 -15909.332} C_VEL
LIN {X 0,Y 308.228,Z 172.755,A -85,B 0,C 180,E1 -15909.611,E2 -15909.611} C_VEL
LIN {X 0,Y 312.012,Z 196.663,A -85,B 0,C 180,E1 -15910.44,E2 -15910.44} C_VEL
LIN {X 0,Y 312.458,Z 201.574,A -85,B 0,C 180,E1 -15910.586,E2 -15910.586} C_VEL
LIN {X 0,Y 311.674,Z 243.351,A -85,B 0,C 180,E1 -15911.57,E2 -15911.57} C_VEL
LIN {X 0,Y 311.173,Z 252.861,A -85,B 0,C 180,E1 -15911.95,E2 -15911.95} C_VEL
LIN {X 0,Y 310.501,Z 262.858,A -85,B 0,C 180,E1 -15912.548,E2 -15912.548} C_VEL
LIN {X 0,Y 309.471,Z 274.217,A -85,B 0,C 180,E1 -15913.509,E2 -15913.509} C_VEL
LIN {X 0,Y 308.567,Z 282.787,A -85,B 0,C 180,E1 -15914.478,E2 -15914.478} C_VEL
LIN {X 0,Y 307.51,Z 290.85,A -85,B 0,C 180,E1 -15915.609,E2 -15915.609} C_VEL
LIN {X 0,Y 306.656,Z 297.513,A -85,B 0,C 180,E1 -15916.751,E2 -15916.751} C_VEL
LIN {X 0,Y 305.872,Z 303.839,A -85,B 0,C 180,E1 -15918.066,E2 -15918.066} C_VEL
LIN {X 0,Y 305.177,Z 309.096,A -85,B 0,C 180,E1 -15919.384,E2 -15919.384} C_VEL
LIN {X 0,Y 304.641,Z 313.479,A -85,B 0,C 180,E1 -15920.707,E2 -15920.707} C_VEL
LIN {X 0,Y 304.066,Z 318.65,A -85,B 0,C 180,E1 -15922.697,E2 -15922.697} C_VEL
LIN {X 0,Y 303.712,Z 322.447,A -85,B 0,C 180,E1 -15924.689,E2 -15924.689} C_VEL
LIN {X 0,Y 303.662,Z 324.192,A -85,B 0,C 180,E1 -15926.019,E2 -15926.019} C_VEL
LIN {X 0,Y 303.599,Z 325.44,A -85,B 0,C 180,E1 -15927.347,E2 -15927.347} C_VEL
LIN {X 0,Y 303.532,Z 326.215,A -85,B 0,C 180,E1 -15928.674,E2 -15928.674} C_VEL
LIN {X 0,Y 303.545,Z 326.509,A -85,B 0,C 180,E1 -15930,E2 -15930} C_VEL
LIN {X 0,Y 303.532,Z 326.209,A -85,B 0,C 180,E1 -15931.327,E2 -15931.327} C_VEL
LIN {X 0,Y 303.599,Z 325.422,A -85,B 0,C 180,E1 -15932.654,E2 -15932.654} C_VEL
LIN {X 0,Y 303.662,Z 324.161,A -85,B 0,C 180,E1 -15933.982,E2 -15933.982} C_VEL
LIN {X 0,Y 303.809,Z 321.392,A -85,B 0,C 180,E1 -15935.893,E2 -15935.893} C_VEL
LIN {X 0,Y 304.064,Z 318.594,A -85,B 0,C 180,E1 -15937.304,E2 -15937.304} C_VEL
LIN {X 0,Y 304.583,Z 313.405,A -85,B 0,C 180,E1 -15939.295,E2 -15939.295} C_VEL
LIN {X 0,Y 305.503,Z 306.568,A -85,B 0,C 180,E1 -15941.277,E2 -15941.277} C_VEL
LIN {X 0,Y 306.44,Z 299.095,A -85,B 0,C 180,E1 -15942.921,E2 -15942.921} C_VEL
LIN {X 0,Y 307.432,Z 291.727,A -85,B 0,C 180,E1 -15944.226,E2 -15944.226} C_VEL
LIN {X 0,Y 308.385,Z 283.835,A -85,B 0,C 180,E1 -15945.363,E2 -15945.363} C_VEL
LIN {X 0,Y 309.325,Z 275.493,A -85,B 0,C 180,E1 -15946.33,E2 -15946.33} C_VEL
LIN {X 0,Y 310.294,Z 264.827,A -85,B 0,C 180,E1 -15947.294,E2 -15947.294} C_VEL
LIN {X 0,Y 311.053,Z 254.021,A -85,B 0,C 180,E1 -15947.972,E2 -15947.972} C_VEL
LIN {X 0,Y 311.601,Z 244.704,A -85,B 0,C 180,E1 -15948.365,E2 -15948.365} C_VEL
LIN {X 0,Y 312.062,Z 221.644,A -85,B 0,C 180,E1 -15948.935,E2 -15948.935} C_VEL
LIN {X 0,Y 312.194,Z 198.546,A -85,B 0,C 180,E1 -15949.478,E2 -15949.478} C_VEL
LIN {X 0,Y 308.445,Z 173.818,A -85,B 0,C 180,E1 -15950.322,E2 -15950.322} C_VEL
LIN {X 0,Y 307.201,Z 166.961,A -85,B 0,C 180,E1 -15950.599,E2 -15950.599} C_VEL
LIN {X 0,Y 307.364,Z 164.92,A -85,B 0,C 180,E1 -15951.109,E2 -15951.109} C_VEL
LIN {X 0,Y 307.955,Z 159.699,A -85,B 0,C 180,E1 -15952.828,E2 -15952.828} C_VEL
LIN {X 0,Y 307.139,Z 153.392,A -85,B 0,C 180,E1 -15955.045,E2 -15955.045} C_VEL
LIN {X 0,Y 305.586,Z 145.345,A -85,B 0,C 180,E1 -15958.037,E2 -15958.037} C_VEL
LIN {X 0,Y 305.445,Z 145.249,A -85,B 0,C 180,E1 -15961.952,E2 -15961.952} C_VEL
LIN {X 0,Y 305.463,Z 145.246,A -85,B 0,C 180,E1 -15965.113,E2 -15965.113} C_VEL
LIN {X 0,Y 305.449,Z 145.241,A -85,B 0,C 180,E1 -15968.529,E2 -15968.529} C_VEL
LIN {X 0,Y 305.455,Z 145.246,A -85,B 0,C 180,E1 -15972.586,E2 -15972.586} C_VEL
LIN {X 0,Y 305.426,Z 145.231,A -85,B 0,C 180,E1 -15976.345,E2 -15976.345} C_VEL
LIN {X 0,Y 305.458,Z 145.248,A -85,B 0,C 180,E1 -15979.893,E2 -15979.893} C_VEL
LIN {X 0,Y 305.482,Z 145.243,A -85,B 0,C 180,E1 -15983.632,E2 -15983.632} C_VEL
LIN {X 0,Y 305.466,Z 145.243,A -85,B 0,C 180,E1 -15986.483,E2 -15986.483} C_VEL
LIN {X 0,Y 305.497,Z 145.242,A -85,B 0,C 180,E1 -15990.95,E2 -15990.95} C_VEL
LIN {X 0,Y 305.573,Z 145.229,A -85,B 0,C 180,E1 -15994.088,E2 -15994.088} C_VEL
LIN {X 0,Y 305.502,Z 145.24,A -85,B 0,C 180,E1 -15998.403,E2 -15998.403} C_VEL
LIN {X 0,Y 305.591,Z 145.227,A -85,B 0,C 180,E1 -16001.218,E2 -16001.218} C_VEL
LIN {X 0,Y 305.65,Z 145.222,A -85,B 0,C 180,E1 -16005.349,E2 -16005.349} C_VEL
LIN {X 0,Y 305.637,Z 145.214,A -85,B 0,C 180,E1 -16009.4,E2 -16009.4} C_VEL
LIN {X 0,Y 305.798,Z 145.202,A -85,B 0,C 180,E1 -16012.074,E2 -16012.074} C_VEL
LIN {X 0,Y 305.687,Z 145.218,A -85,B 0,C 180,E1 -16014.724,E2 -16014.724} C_VEL
LIN {X 0,Y 305.957,Z 145.175,A -85,B 0,C 180,E1 -16018.684,E2 -16018.684} C_VEL
LIN {X 0,Y 305.957,Z 145.18,A -85,B 0,C 180,E1 -16021.316,E2 -16021.316} C_VEL
LIN {X 0,Y 305.854,Z 145.194,A -85,B 0,C 180,E1 -16026.599,E2 -16026.599} C_VEL
LIN {X 0,Y 305.738,Z 145.203,A -85,B 0,C 180,E1 -16029.26,E2 -16029.26} C_VEL
LIN {X 0,Y 305.593,Z 145.231,A -85,B 0,C 180,E1 -16033.296,E2 -16033.296} C_VEL
LIN {X 0,Y 305.596,Z 145.226,A -85,B 0,C 180,E1 -16036.02,E2 -16036.02} C_VEL
LIN {X 0,Y 305.579,Z 145.229,A -85,B 0,C 180,E1 -16039.445,E2 -16039.445} C_VEL
LIN {X 0,Y 305.493,Z 145.245,A -85,B 0,C 180,E1 -16043.042,E2 -16043.042} C_VEL
LIN {X 0,Y 305.528,Z 145.231,A -85,B 0,C 180,E1 -16046.219,E2 -16046.219} C_VEL
LIN {X 0,Y 305.498,Z 145.244,A -85,B 0,C 180,E1 -16049.05,E2 -16049.05} C_VEL
LIN {X 0,Y 305.466,Z 145.239,A -85,B 0,C 180,E1 -16053.517,E2 -16053.517} C_VEL
LIN {X 0,Y 305.476,Z 145.249,A -85,B 0,C 180,E1 -16056.739,E2 -16056.739} C_VEL
LIN {X 0,Y 305.456,Z 145.247,A -85,B 0,C 180,E1 -16060.6,E2 -16060.6} C_VEL
LIN {X 0,Y 305.427,Z 145.251,A -85,B 0,C 180,E1 -16063.655,E2 -16063.655} C_VEL
LIN {X 0,Y 305.456,Z 145.233,A -85,B 0,C 180,E1 -16067.414,E2 -16067.414} C_VEL
LIN {X 0,Y 305.497,Z 145.243,A -85,B 0,C 180,E1 -16071.6,E2 -16071.6} C_VEL
LIN {X 0,Y 305.464,Z 145.234,A -85,B 0,C 180,E1 -16074.887,E2 -16074.887} C_VEL
LIN {X 0,Y 305.454,Z 145.248,A -85,B 0,C 180,E1 -16078.355,E2 -16078.355} C_VEL
LIN {X 0,Y 305.522,Z 145.239,A -85,B 0,C 180,E1 -16081.114,E2 -16081.114} C_VEL
LIN {X 0,Y 305.554,Z 145.303,A -85,B 0,C 180,E1 -16085.18,E2 -16085.18} C_VEL
LIN {X 0,Y 305.678,Z 145.913,A -85,B 0,C 180,E1 -16085.553,E2 -16085.553} C_VEL
LIN {X 0,Y 307.059,Z 153.719,A -85,B 0,C 180,E1 -16088.518,E2 -16088.518} C_VEL
LIN {X 0,Y 307.331,Z 156.457,A -85,B 0,C 180,E1 -16089.421,E2 -16089.421} C_VEL
LIN {X 0,Y 308.322,Z 160.641,A -85,B 0,C 180,E1 -16089.649,E2 -16089.649} C_VEL
LIN {X 0,Y 312.669,Z 183.988,A -85,B 0,C 180,E1 -16090.505,E2 -16090.505} C_VEL
LIN {X 0,Y 311.764,Z 232.627,A -85,B 0,C 180,E1 -16091.645,E2 -16091.645} C_VEL
LIN {X 0,Y 311.351,Z 242.429,A -85,B 0,C 180,E1 -16092.045,E2 -16092.045} C_VEL
LIN {X 0,Y 310.723,Z 253.524,A -85,B 0,C 180,E1 -16092.73,E2 -16092.73} C_VEL
LIN {X 0,Y 309.742,Z 264.346,A -85,B 0,C 180,E1 -16093.693,E2 -16093.693} C_VEL
LIN {X 0,Y 308.844,Z 272.739,A -85,B 0,C 180,E1 -16094.66,E2 -16094.66} C_VEL
LIN {X 0,Y 308.004,Z 280.661,A -85,B 0,C 180,E1 -16095.801,E2 -16095.801} C_VEL
LIN {X 0,Y 307.012,Z 288.049,A -85,B 0,C 180,E1 -16097.103,E2 -16097.103} C_VEL
LIN {X 0,Y 306.007,Z 295.531,A -85,B 0,C 180,E1 -16098.742,E2 -16098.742} C_VEL
LIN {X 0,Y 305.068,Z 302.391,A -85,B 0,C 180,E1 -16100.72,E2 -16100.72} C_VEL
LIN {X 0,Y 304.656,Z 306.06,A -85,B 0,C 180,E1 -16102.044,E2 -16102.044} C_VEL
LIN {X 0,Y 304.145,Z 310.048,A -85,B 0,C 180,E1 -16103.925,E2 -16103.925} C_VEL
LIN {X 0,Y 303.845,Z 313.142,A -85,B 0,C 180,E1 -16106.021,E2 -16106.021} C_VEL
LIN {X 0,Y 303.665,Z 314.415,A -85,B 0,C 180,E1 -16107.347,E2 -16107.347} C_VEL
LIN {X 0,Y 303.561,Z 315.218,A -85,B 0,C 180,E1 -16108.673,E2 -16108.673} C_VEL
LIN {X 0,Y 303.55,Z 315.523,A -85,B 0,C 180,E1 -16110,E2 -16110} C_VEL
LIN {X 0,Y 303.56,Z 315.246,A -85,B 0,C 180,E1 -16111.326,E2 -16111.326} C_VEL
LIN {X 0,Y 303.664,Z 314.498,A -85,B 0,C 180,E1 -16112.653,E2 -16112.653} C_VEL
LIN {X 0,Y 303.84,Z 313.282,A -85,B 0,C 180,E1 -16113.979,E2 -16113.979} C_VEL
LIN {X 0,Y 304.044,Z 311.576,A -85,B 0,C 180,E1 -16115.305,E2 -16115.305} C_VEL
LIN {X 0,Y 304.426,Z 307.833,A -85,B 0,C 180,E1 -16117.294,E2 -16117.294} C_VEL
LIN {X 0,Y 305.027,Z 302.722,A -85,B 0,C 180,E1 -16119.281,E2 -16119.281} C_VEL
LIN {X 0,Y 305.778,Z 297.222,A -85,B 0,C 180,E1 -16120.93,E2 -16120.93} C_VEL
LIN {X 0,Y 306.742,Z 290.31,A -85,B 0,C 180,E1 -16122.571,E2 -16122.571} C_VEL
LIN {X 0,Y 307.756,Z 282.373,A -85,B 0,C 180,E1 -16124.042,E2 -16124.042} C_VEL
LIN {X 0,Y 308.681,Z 274.803,A -85,B 0,C 180,E1 -16125.178,E2 -16125.178} C_VEL
LIN {X 0,Y 309.614,Z 266.867,A -85,B 0,C 180,E1 -16126.144,E2 -16126.144} C_VEL
LIN {X 0,Y 310.346,Z 258.67,A -85,B 0,C 180,E1 -16126.951,E2 -16126.951} C_VEL
LIN {X 0,Y 311.011,Z 250.358,A -85,B 0,C 180,E1 -16127.592,E2 -16127.592} C_VEL
LIN {X 0,Y 311.534,Z 241.369,A -85,B 0,C 180,E1 -16128.113,E2 -16128.113} C_VEL
LIN {X 0,Y 311.874,Z 232.508,A -85,B 0,C 180,E1 -16128.467,E2 -16128.467} C_VEL
LIN {X 0,Y 312.704,Z 184.186,A -85,B 0,C 180,E1 -16129.604,E2 -16129.604} C_VEL
LIN {X 0,Y 308.418,Z 161.063,A -85,B 0,C 180,E1 -16130.451,E2 -16130.451} C_VEL
LIN {X 0,Y 307.29,Z 156.517,A -85,B 0,C 180,E1 -16130.692,E2 -16130.692} C_VEL
LIN {X 0,Y 307.071,Z 154.049,A -85,B 0,C 180,E1 -16131.481,E2 -16131.481} C_VEL
LIN {X 0,Y 305.744,Z 146.235,A -85,B 0,C 180,E1 -16134.441,E2 -16134.441} C_VEL
LIN {X 0,Y 305.565,Z 145.319,A -85,B 0,C 180,E1 -16134.909,E2 -16134.909} C_VEL
LIN {X 0,Y 305.496,Z 145.242,A -85,B 0,C 180,E1 -16139.049,E2 -16139.049} C_VEL
LIN {X 0,Y 305.445,Z 145.25,A -85,B 0,C 180,E1 -16141.952,E2 -16141.952} C_VEL
LIN {X 0,Y 305.462,Z 145.235,A -85,B 0,C 180,E1 -16145.113,E2 -16145.113} C_VEL
LIN {X 0,Y 305.467,Z 145.246,A -85,B 0,C 180,E1 -16148.532,E2 -16148.532} C_VEL
LIN {X 0,Y 305.454,Z 145.229,A -85,B 0,C 180,E1 -16152.585,E2 -16152.585} C_VEL
LIN {X 0,Y 305.425,Z 145.251,A -85,B 0,C 180,E1 -16156.345,E2 -16156.345} C_VEL
LIN {X 0,Y 305.457,Z 145.244,A -85,B 0,C 180,E1 -16159.892,E2 -16159.892} C_VEL
LIN {X 0,Y 305.48,Z 145.245,A -85,B 0,C 180,E1 -16163.631,E2 -16163.631} C_VEL
LIN {X 0,Y 305.459,Z 145.247,A -85,B 0,C 180,E1 -16164.828,E2 -16164.828} C_VEL
LIN {X 0,Y 304.831,Z 145.331,A -85,B 0,C 180,E1 -16165.929,E2 -16165.929} C_VEL
LIN {X 0,Y 302.004,Z 145.69,A -85,B 0,C 180,E1 -16167.721,E2 -16167.721} C_VEL
LIN {X 0,Y 299.576,Z 145.99,A -85,B 0,C 180,E1 -16169.175,E2 -16169.175} C_VEL
LIN {X 0,Y 298.521,Z 146.114,A -85,B 0,C 180,E1 -16170.3,E2 -16170.3} C_VEL
LIN {X 0,Y 298.429,Z 146.122,A -85,B 0,C 180,E1 -16170.682,E2 -16170.682} C_VEL
LIN {X 0,Y 298.476,Z 146.11,A -85,B 0,C 180,E1 -16173.476,E2 -16173.476} C_VEL
LIN {X 0,Y 298.434,Z 146.123,A -85,B 0,C 180,E1 -16176.697,E2 -16176.697} C_VEL
LIN {X 0,Y 298.538,Z 146.103,A -85,B 0,C 180,E1 -16180.757,E2 -16180.757} C_VEL
LIN {X 0,Y 298.592,Z 146.102,A -85,B 0,C 180,E1 -16184.995,E2 -16184.995} C_VEL
LIN {X 0,Y 298.594,Z 146.097,A -85,B 0,C 180,E1 -16189.147,E2 -16189.147} C_VEL
LIN {X 0,Y 298.757,Z 146.072,A -85,B 0,C 180,E1 -16191.886,E2 -16191.886} C_VEL
LIN {X 0,Y 298.659,Z 146.094,A -85,B 0,C 180,E1 -16194.599,E2 -16194.599} C_VEL
LIN {X 0,Y 298.922,Z 146.056,A -85,B 0,C 180,E1 -16198.653,E2 -16198.653} C_VEL
LIN {X 0,Y 298.922,Z 146.05,A -85,B 0,C 180,E1 -16201.347,E2 -16201.347} C_VEL
LIN {X 0,Y 298.798,Z 146.075,A -85,B 0,C 180,E1 -16206.754,E2 -16206.754} C_VEL
LIN {X 0,Y 298.679,Z 146.085,A -85,B 0,C 180,E1 -16209.48,E2 -16209.48} C_VEL
LIN {X 0,Y 298.55,Z 146.11,A -85,B 0,C 180,E1 -16213.615,E2 -16213.615} C_VEL
LIN {X 0,Y 298.547,Z 146.106,A -85,B 0,C 180,E1 -16216.409,E2 -16216.409} C_VEL
LIN {X 0,Y 298.51,Z 146.106,A -85,B 0,C 180,E1 -16219.655,E2 -16219.655} C_VEL
LIN {X 0,Y 298.456,Z 146.119,A -85,B 0,C 180,E1 -16223.598,E2 -16223.598} C_VEL
LIN {X 0,Y 298.49,Z 146.113,A -85,B 0,C 180,E1 -16226.574,E2 -16226.574} C_VEL
LIN {X 0,Y 298.419,Z 146.122,A -85,B 0,C 180,E1 -16229.641,E2 -16229.641} C_VEL
LIN {X 0,Y 298.393,Z 146.127,A -85,B 0,C 180,E1 -16232.8,E2 -16232.8} C_VEL
LIN {X 0,Y 298.444,Z 146.123,A -85,B 0,C 180,E1 -16236.808,E2 -16236.808} C_VEL
LIN {X 0,Y 298.385,Z 146.119,A -85,B 0,C 180,E1 -16241.088,E2 -16241.088} C_VEL
LIN {X 0,Y 298.397,Z 146.105,A -85,B 0,C 180,E1 -16243.103,E2 -16243.103} C_VEL
LIN {X 0,Y 298.401,Z 146.125,A -85,B 0,C 180,E1 -16246.921,E2 -16246.921} C_VEL
LIN {X 0,Y 298.397,Z 146.118,A -85,B 0,C 180,E1 -16251.008,E2 -16251.008} C_VEL
LIN {X 0,Y 298.417,Z 146.126,A -85,B 0,C 180,E1 -16253.93,E2 -16253.93} C_VEL
LIN {X 0,Y 298.395,Z 146.126,A -85,B 0,C 180,E1 -16257.983,E2 -16257.983} C_VEL
LIN {X 0,Y 298.525,Z 146.29,A -85,B 0,C 180,E1 -16261.624,E2 -16261.624} C_VEL
LIN {X 0,Y 300.104,Z 154.393,A -85,B 0,C 180,E1 -16264.699,E2 -16264.699} C_VEL
LIN {X 0,Y 300.995,Z 160.696,A -85,B 0,C 180,E1 -16266.978,E2 -16266.978} C_VEL
LIN {X 0,Y 300.367,Z 166.322,A -85,B 0,C 180,E1 -16268.816,E2 -16268.816} C_VEL
LIN {X 0,Y 300.879,Z 169.825,A -85,B 0,C 180,E1 -16269.019,E2 -16269.019} C_VEL
LIN {X 0,Y 304.868,Z 194.156,A -85,B 0,C 180,E1 -16269.904,E2 -16269.904} C_VEL
LIN {X 0,Y 305.754,Z 203.035,A -85,B 0,C 180,E1 -16270.181,E2 -16270.181} C_VEL
LIN {X 0,Y 304.954,Z 243.331,A -85,B 0,C 180,E1 -16271.152,E2 -16271.152} C_VEL
LIN {X 0,Y 304.448,Z 252.743,A -85,B 0,C 180,E1 -16271.538,E2 -16271.538} C_VEL
LIN {X 0,Y 303.729,Z 262.737,A -85,B 0,C 180,E1 -16272.146,E2 -16272.146} C_VEL
LIN {X 0,Y 302.681,Z 274.093,A -85,B 0,C 180,E1 -16273.128,E2 -16273.128} C_VEL
LIN {X 0,Y 301.736,Z 282.663,A -85,B 0,C 180,E1 -16274.117,E2 -16274.117} C_VEL
LIN {X 0,Y 300.63,Z 290.725,A -85,B 0,C 180,E1 -16275.272,E2 -16275.272} C_VEL
LIN {X 0,Y 299.733,Z 297.387,A -85,B 0,C 180,E1 -16276.44,E2 -16276.44} C_VEL
LIN {X 0,Y 298.915,Z 303.713,A -85,B 0,C 180,E1 -16277.784,E2 -16277.784} C_VEL
LIN {X 0,Y 298.184,Z 308.969,A -85,B 0,C 180,E1 -16279.132,E2 -16279.132} C_VEL
LIN {X 0,Y 297.614,Z 313.352,A -85,B 0,C 180,E1 -16280.486,E2 -16280.486} C_VEL
LIN {X 0,Y 297.005,Z 318.523,A -85,B 0,C 180,E1 -16282.522,E2 -16282.522} C_VEL
LIN {X 0,Y 296.639,Z 322.319,A -85,B 0,C 180,E1 -16284.562,E2 -16284.562} C_VEL
LIN {X 0,Y 296.562,Z 324.064,A -85,B 0,C 180,E1 -16285.923,E2 -16285.923} C_VEL
LIN {X 0,Y 296.528,Z 325.313,A -85,B 0,C 180,E1 -16287.283,E2 -16287.283} C_VEL
LIN {X 0,Y 296.454,Z 326.087,A -85,B 0,C 180,E1 -16288.642,E2 -16288.642} C_VEL
LIN {X 0,Y 296.462,Z 326.38,A -85,B 0,C 180,E1 -16290,E2 -16290} C_VEL
LIN {X 0,Y 296.454,Z 326.081,A -85,B 0,C 180,E1 -16291.359,E2 -16291.359} C_VEL
LIN {X 0,Y 296.528,Z 325.294,A -85,B 0,C 180,E1 -16292.717,E2 -16292.717} C_VEL
LIN {X 0,Y 296.562,Z 324.032,A -85,B 0,C 180,E1 -16294.077,E2 -16294.077} C_VEL
LIN {X 0,Y 296.687,Z 321.683,A -85,B 0,C 180,E1 -16295.786,E2 -16295.786} C_VEL
LIN {X 0,Y 297,Z 318.464,A -85,B 0,C 180,E1 -16297.478,E2 -16297.478} C_VEL
LIN {X 0,Y 297.576,Z 313.275,A -85,B 0,C 180,E1 -16299.516,E2 -16299.516} C_VEL
LIN {X 0,Y 298.521,Z 306.437,A -85,B 0,C 180,E1 -16301.544,E2 -16301.544} C_VEL
LIN {X 0,Y 299.517,Z 298.964,A -85,B 0,C 180,E1 -16303.225,E2 -16303.225} C_VEL
LIN {X 0,Y 300.525,Z 291.595,A -85,B 0,C 180,E1 -16304.56,E2 -16304.56} C_VEL
LIN {X 0,Y 301.534,Z 283.703,A -85,B 0,C 180,E1 -16305.721,E2 -16305.721} C_VEL
LIN {X 0,Y 302.532,Z 275.361,A -85,B 0,C 180,E1 -16306.707,E2 -16306.707} C_VEL
LIN {X 0,Y 303.512,Z 264.692,A -85,B 0,C 180,E1 -16307.693,E2 -16307.693} C_VEL
LIN {X 0,Y 304.331,Z 253.883,A -85,B 0,C 180,E1 -16308.383,E2 -16308.383} C_VEL
LIN {X 0,Y 304.891,Z 244.561,A -85,B 0,C 180,E1 -16308.784,E2 -16308.784} C_VEL
LIN {X 0,Y 305.367,Z 219.817,A -85,B 0,C 180,E1 -16309.408,E2 -16309.408} C_VEL
LIN {X 0,Y 305.592,Z 200.025,A -85,B 0,C 180,E1 -16309.876,E2 -16309.876} C_VEL
LIN {X 0,Y 302.294,Z 177.991,A -85,B 0,C 180,E1 -16310.647,E2 -16310.647} C_VEL
LIN {X 0,Y 300.354,Z 166.698,A -85,B 0,C 180,E1 -16311.103,E2 -16311.103} C_VEL
LIN {X 0,Y 300.406,Z 165.666,A -85,B 0,C 180,E1 -16311.334,E2 -16311.334} C_VEL
LIN {X 0,Y 300.976,Z 160.61,A -85,B 0,C 180,E1 -16313.025,E2 -16313.025} C_VEL
LIN {X 0,Y 299.937,Z 153.253,A -85,B 0,C 180,E1 -16315.689,E2 -16315.689} C_VEL
LIN {X 0,Y 298.516,Z 146.185,A -85,B 0,C 180,E1 -16318.426,E2 -16318.426} C_VEL
LIN {X 0,Y 298.396,Z 146.118,A -85,B 0,C 180,E1 -16322.8,E2 -16322.8} C_VEL
LIN {X 0,Y 298.447,Z 146.116,A -85,B 0,C 180,E1 -16326.808,E2 -16326.808} C_VEL
LIN {X 0,Y 298.387,Z 146.127,A -85,B 0,C 180,E1 -16331.088,E2 -16331.088} C_VEL
LIN {X 0,Y 298.399,Z 146.125,A -85,B 0,C 180,E1 -16333.104,E2 -16333.104} C_VEL
LIN {X 0,Y 298.403,Z 146.103,A -85,B 0,C 180,E1 -16336.921,E2 -16336.921} C_VEL
LIN {X 0,Y 298.405,Z 146.125,A -85,B 0,C 180,E1 -16341.006,E2 -16341.006} C_VEL
LIN {X 0,Y 298.419,Z 146.12,A -85,B 0,C 180,E1 -16343.93,E2 -16343.93} C_VEL
LIN {X 0,Y 298.396,Z 146.126,A -85,B 0,C 180,E1 -16347.984,E2 -16347.984} C_VEL
LIN {X 0,Y 298.471,Z 146.109,A -85,B 0,C 180,E1 -16351.905,E2 -16351.905} C_VEL
LIN {X 0,Y 298.487,Z 146.116,A -85,B 0,C 180,E1 -16354.924,E2 -16354.924} C_VEL
LIN {X 0,Y 298.452,Z 146.113,A -85,B 0,C 180,E1 -16359.316,E2 -16359.316} C_VEL
LIN {X 0,Y 298.539,Z 146.104,A -85,B 0,C 180,E1 -16362.18,E2 -16362.18} C_VEL
LIN {X 0,Y 298.595,Z 146.103,A -85,B 0,C 180,E1 -16364.995,E2 -16364.995} C_VEL
LIN {X 0,Y 298.593,Z 146.09,A -85,B 0,C 180,E1 -16369.147,E2 -16369.147} C_VEL
LIN {X 0,Y 298.742,Z 146.08,A -85,B 0,C 180,E1 -16371.886,E2 -16371.886} C_VEL
LIN {X 0,Y 298.658,Z 146.095,A -85,B 0,C 180,E1 -16374.599,E2 -16374.599} C_VEL
LIN {X 0,Y 298.924,Z 146.05,A -85,B 0,C 180,E1 -16378.653,E2 -16378.653} C_VEL
LIN {X 0,Y 298.924,Z 146.056,A -85,B 0,C 180,E1 -16381.347,E2 -16381.347} C_VEL
LIN {X 0,Y 298.8,Z 146.072,A -85,B 0,C 180,E1 -16386.754,E2 -16386.754} C_VEL
LIN {X 0,Y 298.683,Z 146.082,A -85,B 0,C 180,E1 -16389.481,E2 -16389.481} C_VEL
LIN {X 0,Y 298.556,Z 146.11,A -85,B 0,C 180,E1 -16393.615,E2 -16393.615} C_VEL
LIN {X 0,Y 298.551,Z 146.102,A -85,B 0,C 180,E1 -16396.409,E2 -16396.409} C_VEL
LIN {X 0,Y 298.514,Z 146.11,A -85,B 0,C 180,E1 -16399.655,E2 -16399.655} C_VEL
LIN {X 0,Y 298.46,Z 146.118,A -85,B 0,C 180,E1 -16403.598,E2 -16403.598} C_VEL
LIN {X 0,Y 298.487,Z 146.109,A -85,B 0,C 180,E1 -16406.575,E2 -16406.575} C_VEL
LIN {X 0,Y 298.423,Z 146.123,A -85,B 0,C 180,E1 -16409.641,E2 -16409.641} C_VEL
LIN {X 0,Y 298.397,Z 146.124,A -85,B 0,C 180,E1 -16412.8,E2 -16412.8} C_VEL
LIN {X 0,Y 298.448,Z 146.124,A -85,B 0,C 180,E1 -16416.808,E2 -16416.808} C_VEL
LIN {X 0,Y 298.389,Z 146.127,A -85,B 0,C 180,E1 -16421.088,E2 -16421.088} C_VEL
LIN {X 0,Y 298.4,Z 146.126,A -85,B 0,C 180,E1 -16423.103,E2 -16423.103} C_VEL
LIN {X 0,Y 298.404,Z 146.11,A -85,B 0,C 180,E1 -16426.921,E2 -16426.921} C_VEL
LIN {X 0,Y 298.417,Z 146.124,A -85,B 0,C 180,E1 -16431.004,E2 -16431.004} C_VEL
LIN {X 0,Y 298.433,Z 146.116,A -85,B 0,C 180,E1 -16433.932,E2 -16433.932} C_VEL
LIN {X 0,Y 298.398,Z 146.13,A -85,B 0,C 180,E1 -16437.983,E2 -16437.983} C_VEL
LIN {X 0,Y 298.465,Z 146.12,A -85,B 0,C 180,E1 -16441.904,E2 -16441.904} C_VEL
LIN {X 0,Y 298.532,Z 146.328,A -85,B 0,C 180,E1 -16445.021,E2 -16445.021} C_VEL
LIN {X 0,Y 299.936,Z 153.85,A -85,B 0,C 180,E1 -16447.981,E2 -16447.981} C_VEL
LIN {X 0,Y 300.302,Z 156.649,A -85,B 0,C 180,E1 -16448.924,E2 -16448.924} C_VEL
LIN {X 0,Y 301.915,Z 162.859,A -85,B 0,C 180,E1 -16449.249,E2 -16449.249} C_VEL
LIN {X 0,Y 305.976,Z 184.689,A -85,B 0,C 180,E1 -16450.074,E2 -16450.074} C_VEL
LIN {X 0,Y 305.046,Z 232.773,A -85,B 0,C 180,E1 -16451.226,E2 -16451.226} C_VEL
LIN {X 0,Y 304.624,Z 242.568,A -85,B 0,C 180,E1 -16451.635,E2 -16451.635} C_VEL
LIN {X 0,Y 303.957,Z 253.66,A -85,B 0,C 180,E1 -16452.333,E2 -16452.333} C_VEL
LIN {X 0,Y 302.938,Z 264.479,A -85,B 0,C 180,E1 -16453.316,E2 -16453.316} C_VEL
LIN {X 0,Y 301.998,Z 272.872,A -85,B 0,C 180,E1 -16454.304,E2 -16454.304} C_VEL
LIN {X 0,Y 301.135,Z 280.793,A -85,B 0,C 180,E1 -16455.47,E2 -16455.47} C_VEL
LIN {X 0,Y 300.347,Z 286.482,A -85,B 0,C 180,E1 -16456.467,E2 -16456.467} C_VEL
LIN {X 0,Y 299.46,Z 292.834,A -85,B 0,C 180,E1 -16457.806,E2 -16457.806} C_VEL
LIN {X 0,Y 298.665,Z 298.114,A -85,B 0,C 180,E1 -16459.149,E2 -16459.149} C_VEL
LIN {X 0,Y 298.063,Z 302.521,A -85,B 0,C 180,E1 -16460.499,E2 -16460.499} C_VEL
LIN {X 0,Y 297.399,Z 307.702,A -85,B 0,C 180,E1 -16462.532,E2 -16462.532} C_VEL
LIN {X 0,Y 297.04,Z 310.541,A -85,B 0,C 180,E1 -16463.995,E2 -16463.995} C_VEL
LIN {X 0,Y 296.767,Z 313.271,A -85,B 0,C 180,E1 -16465.926,E2 -16465.926} C_VEL
LIN {X 0,Y 296.596,Z 314.543,A -85,B 0,C 180,E1 -16467.283,E2 -16467.283} C_VEL
LIN {X 0,Y 296.482,Z 315.346,A -85,B 0,C 180,E1 -16468.641,E2 -16468.641} C_VEL
LIN {X 0,Y 296.468,Z 315.651,A -85,B 0,C 180,E1 -16470,E2 -16470} C_VEL
LIN {X 0,Y 296.482,Z 315.374,A -85,B 0,C 180,E1 -16471.358,E2 -16471.358} C_VEL
LIN {X 0,Y 296.594,Z 314.626,A -85,B 0,C 180,E1 -16472.716,E2 -16472.716} C_VEL
LIN {X 0,Y 296.762,Z 313.41,A -85,B 0,C 180,E1 -16474.074,E2 -16474.074} C_VEL
LIN {X 0,Y 296.959,Z 311.704,A -85,B 0,C 180,E1 -16475.432,E2 -16475.432} C_VEL
LIN {X 0,Y 297.386,Z 307.96,A -85,B 0,C 180,E1 -16477.468,E2 -16477.468} C_VEL
LIN {X 0,Y 298.014,Z 302.849,A -85,B 0,C 180,E1 -16479.501,E2 -16479.501} C_VEL
LIN {X 0,Y 298.815,Z 297.348,A -85,B 0,C 180,E1 -16481.188,E2 -16481.188} C_VEL
LIN {X 0,Y 299.826,Z 290.436,A -85,B 0,C 180,E1 -16482.866,E2 -16482.866} C_VEL
LIN {X 0,Y 300.864,Z 282.498,A -85,B 0,C 180,E1 -16484.37,E2 -16484.37} C_VEL
LIN {X 0,Y 301.833,Z 274.928,A -85,B 0,C 180,E1 -16485.531,E2 -16485.531} C_VEL
LIN {X 0,Y 302.803,Z 266.99,A -85,B 0,C 180,E1 -16486.518,E2 -16486.518} C_VEL
LIN {X 0,Y 303.585,Z 258.791,A -85,B 0,C 180,E1 -16487.341,E2 -16487.341} C_VEL
LIN {X 0,Y 304.255,Z 250.478,A -85,B 0,C 180,E1 -16487.996,E2 -16487.996} C_VEL
LIN {X 0,Y 304.807,Z 241.486,A -85,B 0,C 180,E1 -16488.527,E2 -16488.527} C_VEL
LIN {X 0,Y 305.164,Z 232.141,A -85,B 0,C 180,E1 -16488.904,E2 -16488.904} C_VEL
LIN {X 0,Y 305.883,Z 184.196,A -85,B 0,C 180,E1 -16490.062,E2 -16490.062} C_VEL
LIN {X 0,Y 301.833,Z 162.474,A -85,B 0,C 180,E1 -16490.886,E2 -16490.886} C_VEL
LIN {X 0,Y 300.281,Z 156.679,A -85,B 0,C 180,E1 -16491.193,E2 -16491.193} C_VEL
LIN {X 0,Y 299.978,Z 154.18,A -85,B 0,C 180,E1 -16492.015,E2 -16492.015} C_VEL
LIN {X 0,Y 298.539,Z 146.228,A -85,B 0,C 180,E1 -16495.164,E2 -16495.164} C_VEL
LIN {X 0,Y 298.432,Z 146.122,A -85,B 0,C 180,E1 -16499.385,E2 -16499.385} C_VEL
LIN {X 0,Y 298.396,Z 146.126,A -85,B 0,C 180,E1 -16502.8,E2 -16502.8} C_VEL
LIN {X 0,Y 298.464,Z 146.116,A -85,B 0,C 180,E1 -16506.812,E2 -16506.812} C_VEL
LIN {X 0,Y 298.387,Z 146.122,A -85,B 0,C 180,E1 -16511.087,E2 -16511.087} C_VEL
LIN {X 0,Y 298.398,Z 146.107,A -85,B 0,C 180,E1 -16513.103,E2 -16513.103} C_VEL
LIN {X 0,Y 298.402,Z 146.126,A -85,B 0,C 180,E1 -16516.92,E2 -16516.92} C_VEL
LIN {X 0,Y 298.403,Z 146.122,A -85,B 0,C 180,E1 -16521.006,E2 -16521.006} C_VEL
LIN {X 0,Y 298.417,Z 146.123,A -85,B 0,C 180,E1 -16523.93,E2 -16523.93} C_VEL
LIN {X 0,Y 298.394,Z 146.125,A -85,B 0,C 180,E1 -16527.983,E2 -16527.983} C_VEL
LIN {X 0,Y 298.429,Z 146.122,A -85,B 0,C 180,E1 -16530.682,E2 -16530.682} C_VEL
LIN {X 0,Y 297.762,Z 146.203,A -85,B 0,C 180,E1 -16531.808,E2 -16531.808} C_VEL
LIN {X 0,Y 294.964,Z 146.547,A -85,B 0,C 180,E1 -16533.644,E2 -16533.644} C_VEL
LIN {X 0,Y 292.574,Z 146.85,A -85,B 0,C 180,E1 -16535.133,E2 -16535.133} C_VEL
LIN {X 0,Y 291.515,Z 146.982,A -85,B 0,C 180,E1 -16536.285,E2 -16536.285} C_VEL
LIN {X 0,Y 291.409,Z 146.995,A -85,B 0,C 180,E1 -16536.676,E2 -16536.676} C_VEL
LIN {X 0,Y 291.457,Z 146.988,A -85,B 0,C 180,E1 -16540.27,E2 -16540.27} C_VEL
LIN {X 0,Y 291.554,Z 146.979,A -85,B 0,C 180,E1 -16544.623,E2 -16544.623} C_VEL
LIN {X 0,Y 291.537,Z 146.976,A -85,B 0,C 180,E1 -16548.88,E2 -16548.88} C_VEL
LIN {X 0,Y 291.707,Z 146.948,A -85,B 0,C 180,E1 -16551.688,E2 -16551.688} C_VEL
LIN {X 0,Y 291.629,Z 146.971,A -85,B 0,C 180,E1 -16554.468,E2 -16554.468} C_VEL
LIN {X 0,Y 291.889,Z 146.932,A -85,B 0,C 180,E1 -16558.62,E2 -16558.62} C_VEL
LIN {X 0,Y 291.888,Z 146.925,A -85,B 0,C 180,E1 -16561.38,E2 -16561.38} C_VEL
LIN {X 0,Y 291.746,Z 146.954,A -85,B 0,C 180,E1 -16566.918,E2 -16566.918} C_VEL
LIN {X 0,Y 291.628,Z 146.96,A -85,B 0,C 180,E1 -16569.712,E2 -16569.712} C_VEL
LIN {X 0,Y 291.52,Z 146.983,A -85,B 0,C 180,E1 -16573.95,E2 -16573.95} C_VEL
LIN {X 0,Y 291.485,Z 146.987,A -85,B 0,C 180,E1 -16576.818,E2 -16576.818} C_VEL
LIN {X 0,Y 291.449,Z 146.984,A -85,B 0,C 180,E1 -16579.875,E2 -16579.875} C_VEL
LIN {X 0,Y 291.399,Z 146.998,A -85,B 0,C 180,E1 -16584.205,E2 -16584.205} C_VEL
LIN {X 0,Y 291.424,Z 146.988,A -85,B 0,C 180,E1 -16587.271,E2 -16587.271} C_VEL
LIN {X 0,Y 291.336,Z 147.006,A -85,B 0,C 180,E1 -16590.437,E2 -16590.437} C_VEL
LIN {X 0,Y 291.343,Z 147.001,A -85,B 0,C 180,E1 -16593.698,E2 -16593.698} C_VEL
LIN {X 0,Y 291.374,Z 147.002,A -85,B 0,C 180,E1 -16597.254,E2 -16597.254} C_VEL
LIN {X 0,Y 291.331,Z 147,A -85,B 0,C 180,E1 -16600.643,E2 -16600.643} C_VEL
LIN {X 0,Y 291.287,Z 146.994,A -85,B 0,C 180,E1 -16604.402,E2 -16604.402} C_VEL
LIN {X 0,Y 291.324,Z 147.009,A -85,B 0,C 180,E1 -16608.405,E2 -16608.405} C_VEL
LIN {X 0,Y 291.346,Z 146.995,A -85,B 0,C 180,E1 -16611.158,E2 -16611.158} C_VEL
LIN {X 0,Y 291.36,Z 147.004,A -85,B 0,C 180,E1 -16614.626,E2 -16614.626} C_VEL
LIN {X 0,Y 291.372,Z 146.999,A -85,B 0,C 180,E1 -16617.951,E2 -16617.951} C_VEL
LIN {X 0,Y 291.442,Z 147.048,A -85,B 0,C 180,E1 -16621.165,E2 -16621.165} C_VEL
LIN {X 0,Y 293.1,Z 155.309,A -85,B 0,C 180,E1 -16624.431,E2 -16624.431} C_VEL
LIN {X 0,Y 294.006,Z 161.61,A -85,B 0,C 180,E1 -16626.771,E2 -16626.771} C_VEL
LIN {X 0,Y 293.497,Z 166.243,A -85,B 0,C 180,E1 -16628.305,E2 -16628.305} C_VEL
LIN {X 0,Y 294.291,Z 171.054,A -85,B 0,C 180,E1 -16628.561,E2 -16628.561} C_VEL
LIN {X 0,Y 298.249,Z 195.391,A -85,B 0,C 180,E1 -16629.471,E2 -16629.471} C_VEL
LIN {X 0,Y 299.091,Z 202.151,A -85,B 0,C 180,E1 -16629.701,E2 -16629.701} C_VEL
LIN {X 0,Y 298.264,Z 242.749,A -85,B 0,C 180,E1 -16630.697,E2 -16630.697} C_VEL
LIN {X 0,Y 297.803,Z 251.793,A -85,B 0,C 180,E1 -16631.066,E2 -16631.066} C_VEL
LIN {X 0,Y 297.073,Z 261.405,A -85,B 0,C 180,E1 -16631.643,E2 -16631.643} C_VEL
LIN {X 0,Y 296.053,Z 272.38,A -85,B 0,C 180,E1 -16632.561,E2 -16632.561} C_VEL
LIN {X 0,Y 294.918,Z 282.538,A -85,B 0,C 180,E1 -16633.74,E2 -16633.74} C_VEL
LIN {X 0,Y 293.768,Z 290.599,A -85,B 0,C 180,E1 -16634.92,E2 -16634.92} C_VEL
LIN {X 0,Y 292.824,Z 297.261,A -85,B 0,C 180,E1 -16636.113,E2 -16636.113} C_VEL
LIN {X 0,Y 291.979,Z 303.586,A -85,B 0,C 180,E1 -16637.489,E2 -16637.489} C_VEL
LIN {X 0,Y 291.211,Z 308.842,A -85,B 0,C 180,E1 -16638.868,E2 -16638.868} C_VEL
LIN {X 0,Y 290.609,Z 313.225,A -85,B 0,C 180,E1 -16640.254,E2 -16640.254} C_VEL
LIN {X 0,Y 289.968,Z 318.395,A -85,B 0,C 180,E1 -16642.34,E2 -16642.34} C_VEL
LIN {X 0,Y 289.555,Z 322.191,A -85,B 0,C 180,E1 -16644.429,E2 -16644.429} C_VEL
LIN {X 0,Y 289.466,Z 323.936,A -85,B 0,C 180,E1 -16645.823,E2 -16645.823} C_VEL
LIN {X 0,Y 289.435,Z 325.185,A -85,B 0,C 180,E1 -16647.217,E2 -16647.217} C_VEL
LIN {X 0,Y 289.378,Z 325.959,A -85,B 0,C 180,E1 -16648.609,E2 -16648.609} C_VEL
LIN {X 0,Y 289.382,Z 326.252,A -85,B 0,C 180,E1 -16650,E2 -16650} C_VEL
LIN {X 0,Y 289.378,Z 325.953,A -85,B 0,C 180,E1 -16651.392,E2 -16651.392} C_VEL
LIN {X 0,Y 289.435,Z 325.165,A -85,B 0,C 180,E1 -16652.784,E2 -16652.784} C_VEL
LIN {X 0,Y 289.467,Z 323.903,A -85,B 0,C 180,E1 -16654.177,E2 -16654.177} C_VEL
LIN {X 0,Y 289.682,Z 320.991,A -85,B 0,C 180,E1 -16656.267,E2 -16656.267} C_VEL
LIN {X 0,Y 289.932,Z 318.334,A -85,B 0,C 180,E1 -16657.662,E2 -16657.662} C_VEL
LIN {X 0,Y 290.583,Z 313.145,A -85,B 0,C 180,E1 -16659.747,E2 -16659.747} C_VEL
LIN {X 0,Y 291.555,Z 306.306,A -85,B 0,C 180,E1 -16661.824,E2 -16661.824} C_VEL
LIN {X 0,Y 292.581,Z 298.832,A -85,B 0,C 180,E1 -16663.545,E2 -16663.545} C_VEL
LIN {X 0,Y 293.654,Z 291.463,A -85,B 0,C 180,E1 -16664.909,E2 -16664.909} C_VEL
LIN {X 0,Y 294.7,Z 283.57,A -85,B 0,C 180,E1 -16666.095,E2 -16666.095} C_VEL
LIN {X 0,Y 295.748,Z 275.228,A -85,B 0,C 180,E1 -16667.102,E2 -16667.102} C_VEL
LIN {X 0,Y 296.742,Z 264.557,A -85,B 0,C 180,E1 -16668.111,E2 -16668.111} C_VEL
LIN {X 0,Y 297.626,Z 253.746,A -85,B 0,C 180,E1 -16668.813,E2 -16668.813} C_VEL
LIN {X 0,Y 298.191,Z 244.417,A -85,B 0,C 180,E1 -16669.222,E2 -16669.222} C_VEL
LIN {X 0,Y 298.67,Z 220.257,A -85,B 0,C 180,E1 -16669.846,E2 -16669.846} C_VEL
LIN {X 0,Y 298.807,Z 199.718,A -85,B 0,C 180,E1 -16670.351,E2 -16670.351} C_VEL
LIN {X 0,Y 295.19,Z 176.093,A -85,B 0,C 180,E1 -16671.212,E2 -16671.212} C_VEL
LIN {X 0,Y 293.516,Z 166.561,A -85,B 0,C 180,E1 -16671.619,E2 -16671.619} C_VEL
LIN {X 0,Y 293.559,Z 165.533,A -85,B 0,C 180,E1 -16671.856,E2 -16671.856} C_VEL
LIN {X 0,Y 293.986,Z 161.52,A -85,B 0,C 180,E1 -16673.232,E2 -16673.232} C_VEL
LIN {X 0,Y 292.914,Z 154.175,A -85,B 0,C 180,E1 -16675.966,E2 -16675.966} C_VEL
LIN {X 0,Y 291.44,Z 147.019,A -85,B 0,C 180,E1 -16678.836,E2 -16678.836} C_VEL
LIN {X 0,Y 291.344,Z 146.998,A -85,B 0,C 180,E1 -16682.404,E2 -16682.404} C_VEL
LIN {X 0,Y 291.362,Z 147.004,A -85,B 0,C 180,E1 -16685.374,E2 -16685.374} C_VEL
LIN {X 0,Y 291.353,Z 146.995,A -85,B 0,C 180,E1 -16688.842,E2 -16688.842} C_VEL
LIN {X 0,Y 291.32,Z 147.007,A -85,B 0,C 180,E1 -16692.493,E2 -16692.493} C_VEL
LIN {X 0,Y 291.309,Z 146.984,A -85,B 0,C 180,E1 -16696.367,E2 -16696.367} C_VEL
LIN {X 0,Y 291.382,Z 146.999,A -85,B 0,C 180,E1 -16700.518,E2 -16700.518} C_VEL
LIN {X 0,Y 291.408,Z 146.998,A -85,B 0,C 180,E1 -16702.92,E2 -16702.92} C_VEL
LIN {X 0,Y 291.346,Z 147.001,A -85,B 0,C 180,E1 -16706.302,E2 -16706.302} C_VEL
LIN {X 0,Y 291.388,Z 146.997,A -85,B 0,C 180,E1 -16710.26,E2 -16710.26} C_VEL
LIN {X 0,Y 291.422,Z 146.992,A -85,B 0,C 180,E1 -16714.273,E2 -16714.273} C_VEL
LIN {X 0,Y 291.383,Z 146.999,A -85,B 0,C 180,E1 -16717.3,E2 -16717.3} C_VEL
LIN {X 0,Y 291.459,Z 146.982,A -85,B 0,C 180,E1 -16720.27,E2 -16720.27} C_VEL
LIN {X 0,Y 291.557,Z 146.982,A -85,B 0,C 180,E1 -16724.624,E2 -16724.624} C_VEL
LIN {X 0,Y 291.537,Z 146.97,A -85,B 0,C 180,E1 -16728.881,E2 -16728.881} C_VEL
LIN {X 0,Y 291.689,Z 146.957,A -85,B 0,C 180,E1 -16731.688,E2 -16731.688} C_VEL
LIN {X 0,Y 291.628,Z 146.972,A -85,B 0,C 180,E1 -16734.468,E2 -16734.468} C_VEL
LIN {X 0,Y 291.89,Z 146.925,A -85,B 0,C 180,E1 -16738.62,E2 -16738.62} C_VEL
LIN {X 0,Y 291.89,Z 146.932,A -85,B 0,C 180,E1 -16741.38,E2 -16741.38} C_VEL
LIN {X 0,Y 291.748,Z 146.95,A -85,B 0,C 180,E1 -16746.918,E2 -16746.918} C_VEL
LIN {X 0,Y 291.632,Z 146.96,A -85,B 0,C 180,E1 -16749.712,E2 -16749.712} C_VEL
LIN {X 0,Y 291.525,Z 146.983,A -85,B 0,C 180,E1 -16753.95,E2 -16753.95} C_VEL
LIN {X 0,Y 291.489,Z 146.982,A -85,B 0,C 180,E1 -16756.818,E2 -16756.818} C_VEL
LIN {X 0,Y 291.453,Z 146.988,A -85,B 0,C 180,E1 -16759.875,E2 -16759.875} C_VEL
LIN {X 0,Y 291.402,Z 146.995,A -85,B 0,C 180,E1 -16764.205,E2 -16764.205} C_VEL
LIN {X 0,Y 291.422,Z 146.991,A -85,B 0,C 180,E1 -16767.272,E2 -16767.272} C_VEL
LIN {X 0,Y 291.339,Z 147.006,A -85,B 0,C 180,E1 -16770.437,E2 -16770.437} C_VEL
LIN {X 0,Y 291.346,Z 146.996,A -85,B 0,C 180,E1 -16773.698,E2 -16773.698} C_VEL
LIN {X 0,Y 291.378,Z 147.001,A -85,B 0,C 180,E1 -16777.254,E2 -16777.254} C_VEL
LIN {X 0,Y 291.334,Z 147.005,A -85,B 0,C 180,E1 -16780.642,E2 -16780.642} C_VEL
LIN {X 0,Y 291.292,Z 147.011,A -85,B 0,C 180,E1 -16784.402,E2 -16784.402} C_VEL
LIN {X 0,Y 291.328,Z 146.992,A -85,B 0,C 180,E1 -16788.404,E2 -16788.404} C_VEL
LIN {X 0,Y 291.366,Z 147.002,A -85,B 0,C 180,E1 -16791.16,E2 -16791.16} C_VEL
LIN {X 0,Y 291.387,Z 146.986,A -85,B 0,C 180,E1 -16794.629,E2 -16794.629} C_VEL
LIN {X 0,Y 291.375,Z 147.005,A -85,B 0,C 180,E1 -16797.951,E2 -16797.951} C_VEL
LIN {X 0,Y 291.384,Z 147,A -85,B 0,C 180,E1 -16801.158,E2 -16801.158} C_VEL
LIN {X 0,Y 291.491,Z 147.194,A -85,B 0,C 180,E1 -16804.661,E2 -16804.661} C_VEL
LIN {X 0,Y 293.046,Z 155.764,A -85,B 0,C 180,E1 -16808.103,E2 -16808.103} C_VEL
LIN {X 0,Y 293.254,Z 156.956,A -85,B 0,C 180,E1 -16808.413,E2 -16808.413} C_VEL
LIN {X 0,Y 295.779,Z 166.103,A -85,B 0,C 180,E1 -16808.877,E2 -16808.877} C_VEL
LIN {X 0,Y 299.326,Z 185.976,A -85,B 0,C 180,E1 -16809.641,E2 -16809.641} C_VEL
LIN {X 0,Y 298.349,Z 232.918,A -85,B 0,C 180,E1 -16810.788,E2 -16810.788} C_VEL
LIN {X 0,Y 297.911,Z 242.707,A -85,B 0,C 180,E1 -16811.206,E2 -16811.206} C_VEL
LIN {X 0,Y 297.213,Z 253.796,A -85,B 0,C 180,E1 -16811.919,E2 -16811.919} C_VEL
LIN {X 0,Y 296.153,Z 264.613,A -85,B 0,C 180,E1 -16812.922,E2 -16812.922} C_VEL
LIN {X 0,Y 295.178,Z 273.004,A -85,B 0,C 180,E1 -16813.931,E2 -16813.931} C_VEL
LIN {X 0,Y 294.253,Z 280.925,A -85,B 0,C 180,E1 -16815.122,E2 -16815.122} C_VEL
LIN {X 0,Y 293.461,Z 286.614,A -85,B 0,C 180,E1 -16816.143,E2 -16816.143} C_VEL
LIN {X 0,Y 292.529,Z 292.965,A -85,B 0,C 180,E1 -16817.512,E2 -16817.512} C_VEL
LIN {X 0,Y 291.683,Z 298.245,A -85,B 0,C 180,E1 -16818.886,E2 -16818.886} C_VEL
LIN {X 0,Y 291.052,Z 302.651,A -85,B 0,C 180,E1 -16820.268,E2 -16820.268} C_VEL
LIN {X 0,Y 290.365,Z 307.831,A -85,B 0,C 180,E1 -16822.35,E2 -16822.35} C_VEL
LIN {X 0,Y 290.078,Z 309.913,A -85,B 0,C 180,E1 -16823.388,E2 -16823.388} C_VEL
LIN {X 0,Y 289.898,Z 311.636,A -85,B 0,C 180,E1 -16824.435,E2 -16824.435} C_VEL
LIN {X 0,Y 289.692,Z 313.4,A -85,B 0,C 180,E1 -16825.826,E2 -16825.826} C_VEL
LIN {X 0,Y 289.529,Z 314.672,A -85,B 0,C 180,E1 -16827.217,E2 -16827.217} C_VEL
LIN {X 0,Y 289.406,Z 315.474,A -85,B 0,C 180,E1 -16828.608,E2 -16828.608} C_VEL
LIN {X 0,Y 289.388,Z 315.78,A -85,B 0,C 180,E1 -16830,E2 -16830} C_VEL
LIN {X 0,Y 289.406,Z 315.502,A -85,B 0,C 180,E1 -16831.391,E2 -16831.391} C_VEL
LIN {X 0,Y 289.527,Z 314.754,A -85,B 0,C 180,E1 -16832.782,E2 -16832.782} C_VEL
LIN {X 0,Y 289.686,Z 313.538,A -85,B 0,C 180,E1 -16834.173,E2 -16834.173} C_VEL
LIN {X 0,Y 289.882,Z 311.831,A -85,B 0,C 180,E1 -16835.565,E2 -16835.565} C_VEL
LIN {X 0,Y 290.34,Z 308.087,A -85,B 0,C 180,E1 -16837.65,E2 -16837.65} C_VEL
LIN {X 0,Y 291,Z 302.976,A -85,B 0,C 180,E1 -16839.733,E2 -16839.733} C_VEL
LIN {X 0,Y 291.869,Z 297.474,A -85,B 0,C 180,E1 -16841.458,E2 -16841.458} C_VEL
LIN {X 0,Y 292.899,Z 290.562,A -85,B 0,C 180,E1 -16843.176,E2 -16843.176} C_VEL
LIN {X 0,Y 294.004,Z 282.623,A -85,B 0,C 180,E1 -16844.713,E2 -16844.713} C_VEL
LIN {X 0,Y 294.989,Z 275.052,A -85,B 0,C 180,E1 -16845.901,E2 -16845.901} C_VEL
LIN {X 0,Y 296.015,Z 267.113,A -85,B 0,C 180,E1 -16846.908,E2 -16846.908} C_VEL
LIN {X 0,Y 296.833,Z 258.913,A -85,B 0,C 180,E1 -16847.748,E2 -16847.748} C_VEL
LIN {X 0,Y 297.523,Z 250.598,A -85,B 0,C 180,E1 -16848.417,E2 -16848.417} C_VEL
LIN {X 0,Y 298.107,Z 241.603,A -85,B 0,C 180,E1 -16848.959,E2 -16848.959} C_VEL
LIN {X 0,Y 298.453,Z 232.704,A -85,B 0,C 180,E1 -16849.331,E2 -16849.331} C_VEL
LIN {X 0,Y 299.303,Z 185.523,A -85,B 0,C 180,E1 -16850.492,E2 -16850.492} C_VEL
LIN {X 0,Y 295.226,Z 163.715,A -85,B 0,C 180,E1 -16851.347,E2 -16851.347} C_VEL
LIN {X 0,Y 293.22,Z 156.907,A -85,B 0,C 180,E1 -16851.716,E2 -16851.716} C_VEL
LIN {X 0,Y 293.071,Z 155.794,A -85,B 0,C 180,E1 -16852.006,E2 -16852.006} C_VEL
LIN {X 0,Y 291.509,Z 147.101,A -85,B 0,C 180,E1 -16855.527,E2 -16855.527} C_VEL
LIN {X 0,Y 291.387,Z 146.997,A -85,B 0,C 180,E1 -16859.739,E2 -16859.739} C_VEL
LIN {X 0,Y 291.345,Z 147.001,A -85,B 0,C 180,E1 -16863.698,E2 -16863.698} C_VEL
LIN {X 0,Y 291.393,Z 146.996,A -85,B 0,C 180,E1 -16867.258,E2 -16867.258} C_VEL
LIN {X 0,Y 291.334,Z 147,A -85,B 0,C 180,E1 -16870.642,E2 -16870.642} C_VEL
LIN {X 0,Y 291.29,Z 147.006,A -85,B 0,C 180,E1 -16874.401,E2 -16874.401} C_VEL
LIN {X 0,Y 291.325,Z 147.006,A -85,B 0,C 180,E1 -16878.404,E2 -16878.404} C_VEL
LIN {X 0,Y 291.352,Z 147.001,A -85,B 0,C 180,E1 -16881.158,E2 -16881.158} C_VEL
LIN {X 0,Y 291.36,Z 147.002,A -85,B 0,C 180,E1 -16884.626,E2 -16884.626} C_VEL
LIN {X 0,Y 291.371,Z 147,A -85,B 0,C 180,E1 -16887.95,E2 -16887.95} C_VEL
LIN {X 0,Y 291.381,Z 147.001,A -85,B 0,C 180,E1 -16891.158,E2 -16891.158} C_VEL
LIN {X 0,Y 291.411,Z 146.988,A -85,B 0,C 180,E1 -16894.271,E2 -16894.271} C_VEL
LIN {X 0,Y 291.409,Z 146.995,A -85,B 0,C 180,E1 -16896.676,E2 -16896.676} C_VEL
LIN {X 0,Y 290.702,Z 147.085,A -85,B 0,C 180,E1 -16897.829,E2 -16897.829} C_VEL
LIN {X 0,Y 287.882,Z 147.436,A -85,B 0,C 180,E1 -16899.709,E2 -16899.709} C_VEL
LIN {X 0,Y 285.521,Z 147.728,A -85,B 0,C 180,E1 -16901.234,E2 -16901.234} C_VEL
LIN {X 0,Y 284.508,Z 147.85,A -85,B 0,C 180,E1 -16902.415,E2 -16902.415} C_VEL
LIN {X 0,Y 284.423,Z 147.859,A -85,B 0,C 180,E1 -16902.815,E2 -16902.815} C_VEL
LIN {X 0,Y 284.481,Z 147.859,A -85,B 0,C 180,E1 -16905.697,E2 -16905.697} C_VEL
LIN {X 0,Y 284.566,Z 147.842,A -85,B 0,C 180,E1 -16910.044,E2 -16910.044} C_VEL
LIN {X 0,Y 284.697,Z 147.828,A -85,B 0,C 180,E1 -16912.91,E2 -16912.91} C_VEL
LIN {X 0,Y 284.855,Z 147.808,A -85,B 0,C 180,E1 -16918.586,E2 -16918.586} C_VEL
LIN {X 0,Y 284.854,Z 147.8,A -85,B 0,C 180,E1 -16921.414,E2 -16921.414} C_VEL
LIN {X 0,Y 284.698,Z 147.832,A -85,B 0,C 180,E1 -16927.09,E2 -16927.09} C_VEL
LIN {X 0,Y 284.565,Z 147.837,A -85,B 0,C 180,E1 -16929.955,E2 -16929.955} C_VEL
LIN {X 0,Y 284.48,Z 147.859,A -85,B 0,C 180,E1 -16934.303,E2 -16934.303} C_VEL
LIN {X 0,Y 284.424,Z 147.866,A -85,B 0,C 180,E1 -16937.248,E2 -16937.248} C_VEL
LIN {X 0,Y 284.377,Z 147.863,A -85,B 0,C 180,E1 -16940.242,E2 -16940.242} C_VEL
LIN {X 0,Y 284.368,Z 147.874,A -85,B 0,C 180,E1 -16943.876,E2 -16943.876} C_VEL
LIN {X 0,Y 284.398,Z 147.862,A -85,B 0,C 180,E1 -16947.175,E2 -16947.175} C_VEL
LIN {X 0,Y 284.294,Z 147.884,A -85,B 0,C 180,E1 -16951.274,E2 -16951.274} C_VEL
LIN {X 0,Y 284.339,Z 147.873,A -85,B 0,C 180,E1 -16955.348,E2 -16955.348} C_VEL
LIN {X 0,Y 284.31,Z 147.883,A -85,B 0,C 180,E1 -16958.169,E2 -16958.169} C_VEL
LIN {X 0,Y 284.266,Z 147.868,A -85,B 0,C 180,E1 -16962.124,E2 -16962.124} C_VEL
LIN {X 0,Y 284.253,Z 147.884,A -85,B 0,C 180,E1 -16966.189,E2 -16966.189} C_VEL
LIN {X 0,Y 284.305,Z 147.877,A -85,B 0,C 180,E1 -16970.024,E2 -16970.024} C_VEL
LIN {X 0,Y 284.329,Z 147.877,A -85,B 0,C 180,E1 -16973.614,E2 -16973.614} C_VEL
LIN {X 0,Y 284.307,Z 147.873,A -85,B 0,C 180,E1 -16977.19,E2 -16977.19} C_VEL
LIN {X 0,Y 284.383,Z 147.945,A -85,B 0,C 180,E1 -16980.786,E2 -16980.786} C_VEL
LIN {X 0,Y 286.07,Z 156.225,A -85,B 0,C 180,E1 -16984.147,E2 -16984.147} C_VEL
LIN {X 0,Y 287.033,Z 162.525,A -85,B 0,C 180,E1 -16986.555,E2 -16986.555} C_VEL
LIN {X 0,Y 286.706,Z 166.116,A -85,B 0,C 180,E1 -16987.764,E2 -16987.764} C_VEL
LIN {X 0,Y 287.454,Z 170.786,A -85,B 0,C 180,E1 -16988.021,E2 -16988.021} C_VEL
LIN {X 0,Y 291.548,Z 195.67,A -85,B 0,C 180,E1 -16988.987,E2 -16988.987} C_VEL
LIN {X 0,Y 292.41,Z 203.751,A -85,B 0,C 180,E1 -16989.26,E2 -16989.26} C_VEL
LIN {X 0,Y 291.566,Z 242.731,A -85,B 0,C 180,E1 -16990.238,E2 -16990.238} C_VEL
LIN {X 0,Y 291.027,Z 252.506,A -85,B 0,C 180,E1 -16990.653,E2 -16990.653} C_VEL
LIN {X 0,Y 290.249,Z 262.494,A -85,B 0,C 180,E1 -16991.287,E2 -16991.287} C_VEL
LIN {X 0,Y 289.128,Z 273.845,A -85,B 0,C 180,E1 -16992.312,E2 -16992.312} C_VEL
LIN {X 0,Y 288.11,Z 282.413,A -85,B 0,C 180,E1 -16993.344,E2 -16993.344} C_VEL
LIN {X 0,Y 286.915,Z 290.474,A -85,B 0,C 180,E1 -16994.551,E2 -16994.551} C_VEL
LIN {X 0,Y 285.933,Z 297.135,A -85,B 0,C 180,E1 -16995.772,E2 -16995.772} C_VEL
LIN {X 0,Y 285.031,Z 303.46,A -85,B 0,C 180,E1 -16997.179,E2 -16997.179} C_VEL
LIN {X 0,Y 284.238,Z 308.715,A -85,B 0,C 180,E1 -16998.592,E2 -16998.592} C_VEL
LIN {X 0,Y 283.612,Z 313.098,A -85,B 0,C 180,E1 -17000.011,E2 -17000.011} C_VEL
LIN {X 0,Y 282.912,Z 318.268,A -85,B 0,C 180,E1 -17002.148,E2 -17002.148} C_VEL
LIN {X 0,Y 282.479,Z 322.202,A -85,B 0,C 180,E1 -17004.376,E2 -17004.376} C_VEL
LIN {X 0,Y 282.375,Z 323.808,A -85,B 0,C 180,E1 -17005.718,E2 -17005.718} C_VEL
LIN {X 0,Y 282.345,Z 325.057,A -85,B 0,C 180,E1 -17007.147,E2 -17007.147} C_VEL
LIN {X 0,Y 282.303,Z 325.832,A -85,B 0,C 180,E1 -17008.574,E2 -17008.574} C_VEL
LIN {X 0,Y 282.304,Z 326.124,A -85,B 0,C 180,E1 -17010,E2 -17010} C_VEL
LIN {X 0,Y 282.303,Z 325.825,A -85,B 0,C 180,E1 -17011.427,E2 -17011.427} C_VEL
LIN {X 0,Y 282.345,Z 325.036,A -85,B 0,C 180,E1 -17012.854,E2 -17012.854} C_VEL
LIN {X 0,Y 282.375,Z 323.773,A -85,B 0,C 180,E1 -17014.282,E2 -17014.282} C_VEL
LIN {X 0,Y 282.602,Z 320.86,A -85,B 0,C 180,E1 -17016.426,E2 -17016.426} C_VEL
LIN {X 0,Y 282.886,Z 318.204,A -85,B 0,C 180,E1 -17017.854,E2 -17017.854} C_VEL
LIN {X 0,Y 283.565,Z 313.015,A -85,B 0,C 180,E1 -17019.991,E2 -17019.991} C_VEL
LIN {X 0,Y 284.584,Z 306.175,A -85,B 0,C 180,E1 -17022.118,E2 -17022.118} C_VEL
LIN {X 0,Y 285.669,Z 298.701,A -85,B 0,C 180,E1 -17023.879,E2 -17023.879} C_VEL
LIN {X 0,Y 286.794,Z 291.332,A -85,B 0,C 180,E1 -17025.274,E2 -17025.274} C_VEL
LIN {X 0,Y 287.891,Z 283.438,A -85,B 0,C 180,E1 -17026.487,E2 -17026.487} C_VEL
LIN {X 0,Y 288.964,Z 275.095,A -85,B 0,C 180,E1 -17027.517,E2 -17027.517} C_VEL
LIN {X 0,Y 290.012,Z 264.423,A -85,B 0,C 180,E1 -17028.546,E2 -17028.546} C_VEL
LIN {X 0,Y 290.933,Z 253.608,A -85,B 0,C 180,E1 -17029.262,E2 -17029.262} C_VEL
LIN {X 0,Y 291.524,Z 243.818,A -85,B 0,C 180,E1 -17029.696,E2 -17029.696} C_VEL
LIN {X 0,Y 292.278,Z 206.847,A -85,B 0,C 180,E1 -17030.64,E2 -17030.64} C_VEL
LIN {X 0,Y 292.074,Z 199.672,A -85,B 0,C 180,E1 -17030.839,E2 -17030.839} C_VEL
LIN {X 0,Y 287.949,Z 173.376,A -85,B 0,C 180,E1 -17031.839,E2 -17031.839} C_VEL
LIN {X 0,Y 286.667,Z 166.329,A -85,B 0,C 180,E1 -17032.174,E2 -17032.174} C_VEL
LIN {X 0,Y 287.017,Z 162.433,A -85,B 0,C 180,E1 -17033.447,E2 -17033.447} C_VEL
LIN {X 0,Y 285.855,Z 155.078,A -85,B 0,C 180,E1 -17036.267,E2 -17036.267} C_VEL
LIN {X 0,Y 284.384,Z 147.906,A -85,B 0,C 180,E1 -17039.215,E2 -17039.215} C_VEL
LIN {X 0,Y 284.306,Z 147.871,A -85,B 0,C 180,E1 -17042.945,E2 -17042.945} C_VEL
LIN {X 0,Y 284.333,Z 147.876,A -85,B 0,C 180,E1 -17046.386,E2 -17046.386} C_VEL
LIN {X 0,Y 284.306,Z 147.877,A -85,B 0,C 180,E1 -17049.995,E2 -17049.995} C_VEL
LIN {X 0,Y 284.246,Z 147.881,A -85,B 0,C 180,E1 -17054.191,E2 -17054.191} C_VEL
LIN {X 0,Y 284.272,Z 147.872,A -85,B 0,C 180,E1 -17058.125,E2 -17058.125} C_VEL
LIN {X 0,Y 284.323,Z 147.88,A -85,B 0,C 180,E1 -17062.278,E2 -17062.278} C_VEL
LIN {X 0,Y 284.309,Z 147.877,A -85,B 0,C 180,E1 -17065.351,E2 -17065.351} C_VEL
LIN {X 0,Y 284.297,Z 147.884,A -85,B 0,C 180,E1 -17068.726,E2 -17068.726} C_VEL
LIN {X 0,Y 284.401,Z 147.862,A -85,B 0,C 180,E1 -17072.826,E2 -17072.826} C_VEL
LIN {X 0,Y 284.368,Z 147.876,A -85,B 0,C 180,E1 -17076.707,E2 -17076.707} C_VEL
LIN {X 0,Y 284.405,Z 147.864,A -85,B 0,C 180,E1 -17081.262,E2 -17081.262} C_VEL
LIN {X 0,Y 284.494,Z 147.86,A -85,B 0,C 180,E1 -17084.459,E2 -17084.459} C_VEL
LIN {X 0,Y 284.489,Z 147.848,A -85,B 0,C 180,E1 -17088.602,E2 -17088.602} C_VEL
LIN {X 0,Y 284.64,Z 147.834,A -85,B 0,C 180,E1 -17091.481,E2 -17091.481} C_VEL
LIN {X 0,Y 284.598,Z 147.848,A -85,B 0,C 180,E1 -17094.331,E2 -17094.331} C_VEL
LIN {X 0,Y 284.856,Z 147.8,A -85,B 0,C 180,E1 -17098.586,E2 -17098.586} C_VEL
LIN {X 0,Y 284.856,Z 147.807,A -85,B 0,C 180,E1 -17101.414,E2 -17101.414} C_VEL
LIN {X 0,Y 284.7,Z 147.828,A -85,B 0,C 180,E1 -17107.09,E2 -17107.09} C_VEL
LIN {X 0,Y 284.569,Z 147.841,A -85,B 0,C 180,E1 -17109.955,E2 -17109.955} C_VEL
LIN {X 0,Y 284.485,Z 147.859,A -85,B 0,C 180,E1 -17114.303,E2 -17114.303} C_VEL
LIN {X 0,Y 284.427,Z 147.859,A -85,B 0,C 180,E1 -17117.248,E2 -17117.248} C_VEL
LIN {X 0,Y 284.381,Z 147.868,A -85,B 0,C 180,E1 -17120.242,E2 -17120.242} C_VEL
LIN {X 0,Y 284.371,Z 147.871,A -85,B 0,C 180,E1 -17123.875,E2 -17123.875} C_VEL
LIN {X 0,Y 284.397,Z 147.864,A -85,B 0,C 180,E1 -17127.173,E2 -17127.173} C_VEL
LIN {X 0,Y 284.298,Z 147.883,A -85,B 0,C 180,E1 -17131.274,E2 -17131.274} C_VEL
LIN {X 0,Y 284.343,Z 147.876,A -85,B 0,C 180,E1 -17135.348,E2 -17135.348} C_VEL
LIN {X 0,Y 284.314,Z 147.882,A -85,B 0,C 180,E1 -17138.169,E2 -17138.169} C_VEL
LIN {X 0,Y 284.271,Z 147.887,A -85,B 0,C 180,E1 -17142.124,E2 -17142.124} C_VEL
LIN {X 0,Y 284.257,Z 147.875,A -85,B 0,C 180,E1 -17146.189,E2 -17146.189} C_VEL
LIN {X 0,Y 284.309,Z 147.877,A -85,B 0,C 180,E1 -17150.024,E2 -17150.024} C_VEL
LIN {X 0,Y 284.352,Z 147.871,A -85,B 0,C 180,E1 -17153.617,E2 -17153.617} C_VEL
LIN {X 0,Y 284.31,Z 147.88,A -85,B 0,C 180,E1 -17157.189,E2 -17157.189} C_VEL
LIN {X 0,Y 284.361,Z 147.871,A -85,B 0,C 180,E1 -17160.376,E2 -17160.376} C_VEL
LIN {X 0,Y 284.414,Z 147.99,A -85,B 0,C 180,E1 -17164.23,E2 -17164.23} C_VEL
LIN {X 0,Y 286.03,Z 156.572,A -85,B 0,C 180,E1 -17167.759,E2 -17167.759} C_VEL
LIN {X 0,Y 286.577,Z 158.617,A -85,B 0,C 180,E1 -17167.96,E2 -17167.96} C_VEL
LIN {X 0,Y 289.089,Z 166.97,A -85,B 0,C 180,E1 -17168.383,E2 -17168.383} C_VEL
LIN {X 0,Y 292.685,Z 186.701,A -85,B 0,C 180,E1 -17169.172,E2 -17169.172} C_VEL
LIN {X 0,Y 291.668,Z 233.064,A -85,B 0,C 180,E1 -17170.33,E2 -17170.33} C_VEL
LIN {X 0,Y 291.214,Z 242.847,A -85,B 0,C 180,E1 -17170.757,E2 -17170.757} C_VEL
LIN {X 0,Y 290.49,Z 253.931,A -85,B 0,C 180,E1 -17171.485,E2 -17171.485} C_VEL
LIN {X 0,Y 289.391,Z 264.746,A -85,B 0,C 180,E1 -17172.51,E2 -17172.51} C_VEL
LIN {X 0,Y 288.382,Z 273.136,A -85,B 0,C 180,E1 -17173.542,E2 -17173.542} C_VEL
LIN {X 0,Y 287.371,Z 281.057,A -85,B 0,C 180,E1 -17174.757,E2 -17174.757} C_VEL
LIN {X 0,Y 286.585,Z 286.745,A -85,B 0,C 180,E1 -17175.804,E2 -17175.804} C_VEL
LIN {X 0,Y 285.599,Z 293.096,A -85,B 0,C 180,E1 -17177.204,E2 -17177.204} C_VEL
LIN {X 0,Y 284.719,Z 298.376,A -85,B 0,C 180,E1 -17178.611,E2 -17178.611} C_VEL
LIN {X 0,Y 284.045,Z 302.782,A -85,B 0,C 180,E1 -17180.026,E2 -17180.026} C_VEL
LIN {X 0,Y 283.34,Z 307.961,A -85,B 0,C 180,E1 -17182.159,E2 -17182.159} C_VEL
LIN {X 0,Y 282.962,Z 310.424,A -85,B 0,C 180,E1 -17183.46,E2 -17183.46} C_VEL
LIN {X 0,Y 282.619,Z 313.529,A -85,B 0,C 180,E1 -17185.721,E2 -17185.721} C_VEL
LIN {X 0,Y 282.463,Z 314.8,A -85,B 0,C 180,E1 -17187.147,E2 -17187.147} C_VEL
LIN {X 0,Y 282.332,Z 315.602,A -85,B 0,C 180,E1 -17188.573,E2 -17188.573} C_VEL
LIN {X 0,Y 282.31,Z 315.908,A -85,B 0,C 180,E1 -17190,E2 -17190} C_VEL
LIN {X 0,Y 282.332,Z 315.629,A -85,B 0,C 180,E1 -17191.426,E2 -17191.426} C_VEL
LIN {X 0,Y 282.461,Z 314.881,A -85,B 0,C 180,E1 -17192.852,E2 -17192.852} C_VEL
LIN {X 0,Y 282.613,Z 313.665,A -85,B 0,C 180,E1 -17194.278,E2 -17194.278} C_VEL
LIN {X 0,Y 282.811,Z 311.959,A -85,B 0,C 180,E1 -17195.704,E2 -17195.704} C_VEL
LIN {X 0,Y 283.302,Z 308.215,A -85,B 0,C 180,E1 -17197.842,E2 -17197.842} C_VEL
LIN {X 0,Y 284.007,Z 303.103,A -85,B 0,C 180,E1 -17199.975,E2 -17199.975} C_VEL
LIN {X 0,Y 284.933,Z 297.601,A -85,B 0,C 180,E1 -17201.741,E2 -17201.741} C_VEL
LIN {X 0,Y 285.996,Z 290.687,A -85,B 0,C 180,E1 -17203.5,E2 -17203.5} C_VEL
LIN {X 0,Y 287.157,Z 282.748,A -85,B 0,C 180,E1 -17205.072,E2 -17205.072} C_VEL
LIN {X 0,Y 288.159,Z 275.177,A -85,B 0,C 180,E1 -17206.288,E2 -17206.288} C_VEL
LIN {X 0,Y 289.217,Z 267.237,A -85,B 0,C 180,E1 -17207.318,E2 -17207.318} C_VEL
LIN {X 0,Y 290.102,Z 259.035,A -85,B 0,C 180,E1 -17208.174,E2 -17208.174} C_VEL
LIN {X 0,Y 290.812,Z 250.718,A -85,B 0,C 180,E1 -17208.858,E2 -17208.858} C_VEL
LIN {X 0,Y 291.413,Z 241.72,A -85,B 0,C 180,E1 -17209.412,E2 -17209.412} C_VEL
LIN {X 0,Y 291.786,Z 232.807,A -85,B 0,C 180,E1 -17209.791,E2 -17209.791} C_VEL
LIN {X 0,Y 292.601,Z 185.953,A -85,B 0,C 180,E1 -17210.975,E2 -17210.975} C_VEL
LIN {X 0,Y 288.811,Z 165.678,A -85,B 0,C 180,E1 -17211.796,E2 -17211.796} C_VEL
LIN {X 0,Y 286.11,Z 156.977,A -85,B 0,C 180,E1 -17212.291,E2 -17212.291} C_VEL
LIN {X 0,Y 285.82,Z 155.433,A -85,B 0,C 180,E1 -17212.785,E2 -17212.785} C_VEL
LIN {X 0,Y 284.455,Z 147.971,A -85,B 0,C 180,E1 -17215.912,E2 -17215.912} C_VEL
LIN {X 0,Y 284.315,Z 147.876,A -85,B 0,C 180,E1 -17220.098,E2 -17220.098} C_VEL
LIN {X 0,Y 284.306,Z 147.881,A -85,B 0,C 180,E1 -17222.945,E2 -17222.945} C_VEL
LIN {X 0,Y 284.35,Z 147.87,A -85,B 0,C 180,E1 -17226.383,E2 -17226.383} C_VEL
LIN {X 0,Y 284.306,Z 147.878,A -85,B 0,C 180,E1 -17229.994,E2 -17229.994} C_VEL
LIN {X 0,Y 284.245,Z 147.879,A -85,B 0,C 180,E1 -17234.19,E2 -17234.19} C_VEL
LIN {X 0,Y 284.271,Z 147.886,A -85,B 0,C 180,E1 -17238.124,E2 -17238.124} C_VEL
LIN {X 0,Y 284.321,Z 147.88,A -85,B 0,C 180,E1 -17242.278,E2 -17242.278} C_VEL
LIN {X 0,Y 284.307,Z 147.877,A -85,B 0,C 180,E1 -17245.35,E2 -17245.35} C_VEL
LIN {X 0,Y 284.295,Z 147.882,A -85,B 0,C 180,E1 -17248.725,E2 -17248.725} C_VEL
LIN {X 0,Y 284.394,Z 147.865,A -85,B 0,C 180,E1 -17252.827,E2 -17252.827} C_VEL
LIN {X 0,Y 284.365,Z 147.875,A -85,B 0,C 180,E1 -17256.707,E2 -17256.707} C_VEL
LIN {X 0,Y 284.402,Z 147.858,A -85,B 0,C 180,E1 -17261.261,E2 -17261.261} C_VEL
LIN {X 0,Y 284.423,Z 147.859,A -85,B 0,C 180,E1 -17262.815,E2 -17262.815} C_VEL
LIN {X 0,Y 283.746,Z 147.948,A -85,B 0,C 180,E1 -17263.997,E2 -17263.997} C_VEL
LIN {X 0,Y 280.891,Z 148.307,A -85,B 0,C 180,E1 -17265.924,E2 -17265.924} C_VEL
LIN {X 0,Y 278.5,Z 148.603,A -85,B 0,C 180,E1 -17267.489,E2 -17267.489} C_VEL
LIN {X 0,Y 277.512,Z 148.724,A -85,B 0,C 180,E1 -17268.702,E2 -17268.702} C_VEL
LIN {X 0,Y 277.451,Z 148.729,A -85,B 0,C 180,E1 -17269.113,E2 -17269.113} C_VEL
LIN {X 0,Y 277.614,Z 148.701,A -85,B 0,C 180,E1 -17271.263,E2 -17271.263} C_VEL
LIN {X 0,Y 277.571,Z 148.72,A -85,B 0,C 180,E1 -17274.187,E2 -17274.187} C_VEL
LIN {X 0,Y 277.82,Z 148.684,A -85,B 0,C 180,E1 -17278.55,E2 -17278.55} C_VEL
LIN {X 0,Y 277.82,Z 148.675,A -85,B 0,C 180,E1 -17281.449,E2 -17281.449} C_VEL
LIN {X 0,Y 277.653,Z 148.711,A -85,B 0,C 180,E1 -17287.271,E2 -17287.271} C_VEL
LIN {X 0,Y 277.505,Z 148.714,A -85,B 0,C 180,E1 -17290.211,E2 -17290.211} C_VEL
LIN {X 0,Y 277.433,Z 148.737,A -85,B 0,C 180,E1 -17294.674,E2 -17294.674} C_VEL
LIN {X 0,Y 277.343,Z 148.739,A -85,B 0,C 180,E1 -17299.234,E2 -17299.234} C_VEL
LIN {X 0,Y 277.318,Z 148.752,A -85,B 0,C 180,E1 -17304.171,E2 -17304.171} C_VEL
LIN {X 0,Y 277.326,Z 148.741,A -85,B 0,C 180,E1 -17307.506,E2 -17307.506} C_VEL
LIN {X 0,Y 277.27,Z 148.758,A -85,B 0,C 180,E1 -17310.481,E2 -17310.481} C_VEL
LIN {X 0,Y 277.245,Z 148.757,A -85,B 0,C 180,E1 -17313.896,E2 -17313.896} C_VEL
LIN {X 0,Y 277.266,Z 148.759,A -85,B 0,C 180,E1 -17317.469,E2 -17317.469} C_VEL
LIN {X 0,Y 277.207,Z 148.755,A -85,B 0,C 180,E1 -17321.237,E2 -17321.237} C_VEL
LIN {X 0,Y 277.198,Z 148.757,A -85,B 0,C 180,E1 -17325.227,E2 -17325.227} C_VEL
LIN {X 0,Y 277.221,Z 148.764,A -85,B 0,C 180,E1 -17329.512,E2 -17329.512} C_VEL
LIN {X 0,Y 277.263,Z 148.749,A -85,B 0,C 180,E1 -17332.531,E2 -17332.531} C_VEL
LIN {X 0,Y 277.246,Z 148.755,A -85,B 0,C 180,E1 -17336.105,E2 -17336.105} C_VEL
LIN {X 0,Y 277.344,Z 148.841,A -85,B 0,C 180,E1 -17340.388,E2 -17340.388} C_VEL
LIN {X 0,Y 279.041,Z 157.136,A -85,B 0,C 180,E1 -17343.848,E2 -17343.848} C_VEL
LIN {X 0,Y 280.022,Z 163.438,A -85,B 0,C 180,E1 -17346.324,E2 -17346.324} C_VEL
LIN {X 0,Y 279.882,Z 165.987,A -85,B 0,C 180,E1 -17347.192,E2 -17347.192} C_VEL
LIN {X 0,Y 280.677,Z 170.772,A -85,B 0,C 180,E1 -17347.464,E2 -17347.464} C_VEL
LIN {X 0,Y 284.847,Z 195.771,A -85,B 0,C 180,E1 -17348.474,E2 -17348.474} C_VEL
LIN {X 0,Y 285.795,Z 203.575,A -85,B 0,C 180,E1 -17348.755,E2 -17348.755} C_VEL
LIN {X 0,Y 284.902,Z 242.676,A -85,B 0,C 180,E1 -17349.758,E2 -17349.758} C_VEL
LIN {X 0,Y 284.33,Z 252.483,A -85,B 0,C 180,E1 -17350.184,E2 -17350.184} C_VEL
LIN {X 0,Y 283.436,Z 263.59,A -85,B 0,C 180,E1 -17350.915,E2 -17350.915} C_VEL
LIN {X 0,Y 282.377,Z 273.721,A -85,B 0,C 180,E1 -17351.874,E2 -17351.874} C_VEL
LIN {X 0,Y 281.307,Z 282.288,A -85,B 0,C 180,E1 -17352.93,E2 -17352.93} C_VEL
LIN {X 0,Y 280.08,Z 290.348,A -85,B 0,C 180,E1 -17354.164,E2 -17354.164} C_VEL
LIN {X 0,Y 279.057,Z 297.009,A -85,B 0,C 180,E1 -17355.413,E2 -17355.413} C_VEL
LIN {X 0,Y 278.089,Z 303.333,A -85,B 0,C 180,E1 -17356.853,E2 -17356.853} C_VEL
LIN {X 0,Y 277.252,Z 308.588,A -85,B 0,C 180,E1 -17358.3,E2 -17358.3} C_VEL
LIN {X 0,Y 276.596,Z 312.97,A -85,B 0,C 180,E1 -17359.755,E2 -17359.755} C_VEL
LIN {X 0,Y 275.883,Z 318.14,A -85,B 0,C 180,E1 -17361.946,E2 -17361.946} C_VEL
LIN {X 0,Y 275.416,Z 321.936,A -85,B 0,C 180,E1 -17364.142,E2 -17364.142} C_VEL
LIN {X 0,Y 275.288,Z 323.68,A -85,B 0,C 180,E1 -17365.608,E2 -17365.608} C_VEL
LIN {X 0,Y 275.257,Z 324.929,A -85,B 0,C 180,E1 -17367.073,E2 -17367.073} C_VEL
LIN {X 0,Y 275.23,Z 325.704,A -85,B 0,C 180,E1 -17368.537,E2 -17368.537} C_VEL
LIN {X 0,Y 275.228,Z 325.996,A -85,B 0,C 180,E1 -17370,E2 -17370} C_VEL
LIN {X 0,Y 275.23,Z 325.697,A -85,B 0,C 180,E1 -17371.464,E2 -17371.464} C_VEL
LIN {X 0,Y 275.257,Z 324.907,A -85,B 0,C 180,E1 -17372.927,E2 -17372.927} C_VEL
LIN {X 0,Y 275.396,Z 322.301,A -85,B 0,C 180,E1 -17375.579,E2 -17375.579} C_VEL
LIN {X 0,Y 275.693,Z 319.557,A -85,B 0,C 180,E1 -17377.323,E2 -17377.323} C_VEL
LIN {X 0,Y 276.262,Z 314.803,A -85,B 0,C 180,E1 -17379.518,E2 -17379.518} C_VEL
LIN {X 0,Y 277.061,Z 309.657,A -85,B 0,C 180,E1 -17381.338,E2 -17381.338} C_VEL
LIN {X 0,Y 277.87,Z 304.628,A -85,B 0,C 180,E1 -17382.786,E2 -17382.786} C_VEL
LIN {X 0,Y 278.777,Z 298.57,A -85,B 0,C 180,E1 -17384.229,E2 -17384.229} C_VEL
LIN {X 0,Y 279.944,Z 291.2,A -85,B 0,C 180,E1 -17385.657,E2 -17385.657} C_VEL
LIN {X 0,Y 281.096,Z 283.306,A -85,B 0,C 180,E1 -17386.897,E2 -17386.897} C_VEL
LIN {X 0,Y 282.201,Z 274.962,A -85,B 0,C 180,E1 -17387.95,E2 -17387.95} C_VEL
LIN {X 0,Y 283.294,Z 264.331,A -85,B 0,C 180,E1 -17388.999,E2 -17388.999} C_VEL
LIN {X 0,Y 284.281,Z 253.009,A -85,B 0,C 180,E1 -17389.758,E2 -17389.758} C_VEL
LIN {X 0,Y 284.847,Z 244.083,A -85,B 0,C 180,E1 -17390.162,E2 -17390.162} C_VEL
LIN {X 0,Y 285.481,Z 214.869,A -85,B 0,C 180,E1 -17390.939,E2 -17390.939} C_VEL
LIN {X 0,Y 285.516,Z 201.108,A -85,B 0,C 180,E1 -17391.299,E2 -17391.299} C_VEL
LIN {X 0,Y 281.539,Z 175.411,A -85,B 0,C 180,E1 -17392.304,E2 -17392.304} C_VEL
LIN {X 0,Y 279.867,Z 166.293,A -85,B 0,C 180,E1 -17392.73,E2 -17392.73} C_VEL
LIN {X 0,Y 279.919,Z 165.266,A -85,B 0,C 180,E1 -17392.981,E2 -17392.981} C_VEL
LIN {X 0,Y 279.773,Z 161.48,A -85,B 0,C 180,E1 -17394.398,E2 -17394.398} C_VEL
LIN {X 0,Y 278.229,Z 152.828,A -85,B 0,C 180,E1 -17397.86,E2 -17397.86} C_VEL
LIN {X 0,Y 277.345,Z 148.793,A -85,B 0,C 180,E1 -17399.613,E2 -17399.613} C_VEL
LIN {X 0,Y 277.248,Z 148.754,A -85,B 0,C 180,E1 -17403.896,E2 -17403.896} C_VEL
LIN {X 0,Y 277.268,Z 148.747,A -85,B 0,C 180,E1 -17407.47,E2 -17407.47} C_VEL
LIN {X 0,Y 277.21,Z 148.765,A -85,B 0,C 180,E1 -17411.237,E2 -17411.237} C_VEL
LIN {X 0,Y 277.201,Z 148.747,A -85,B 0,C 180,E1 -17415.227,E2 -17415.227} C_VEL
LIN {X 0,Y 277.223,Z 148.758,A -85,B 0,C 180,E1 -17419.513,E2 -17419.513} C_VEL
LIN {X 0,Y 277.268,Z 148.758,A -85,B 0,C 180,E1 -17422.531,E2 -17422.531} C_VEL
LIN {X 0,Y 277.248,Z 148.757,A -85,B 0,C 180,E1 -17426.105,E2 -17426.105} C_VEL
LIN {X 0,Y 277.262,Z 148.759,A -85,B 0,C 180,E1 -17429.539,E2 -17429.539} C_VEL
LIN {X 0,Y 277.362,Z 148.738,A -85,B 0,C 180,E1 -17432.865,E2 -17432.865} C_VEL
LIN {X 0,Y 277.331,Z 148.75,A -85,B 0,C 180,E1 -17436.08,E2 -17436.08} C_VEL
LIN {X 0,Y 277.347,Z 148.739,A -85,B 0,C 180,E1 -17440.766,E2 -17440.766} C_VEL
LIN {X 0,Y 277.436,Z 148.737,A -85,B 0,C 180,E1 -17445.326,E2 -17445.326} C_VEL
LIN {X 0,Y 277.463,Z 148.719,A -85,B 0,C 180,E1 -17449.787,E2 -17449.787} C_VEL
LIN {X 0,Y 277.642,Z 148.712,A -85,B 0,C 180,E1 -17452.729,E2 -17452.729} C_VEL
LIN {X 0,Y 277.822,Z 148.675,A -85,B 0,C 180,E1 -17458.551,E2 -17458.551} C_VEL
LIN {X 0,Y 277.822,Z 148.683,A -85,B 0,C 180,E1 -17461.45,E2 -17461.45} C_VEL
LIN {X 0,Y 277.655,Z 148.706,A -85,B 0,C 180,E1 -17467.271,E2 -17467.271} C_VEL
LIN {X 0,Y 277.509,Z 148.722,A -85,B 0,C 180,E1 -17470.211,E2 -17470.211} C_VEL
LIN {X 0,Y 277.437,Z 148.736,A -85,B 0,C 180,E1 -17474.674,E2 -17474.674} C_VEL
LIN {X 0,Y 277.347,Z 148.738,A -85,B 0,C 180,E1 -17479.234,E2 -17479.234} C_VEL
LIN {X 0,Y 277.321,Z 148.749,A -85,B 0,C 180,E1 -17484.17,E2 -17484.17} C_VEL
LIN {X 0,Y 277.326,Z 148.746,A -85,B 0,C 180,E1 -17487.505,E2 -17487.505} C_VEL
LIN {X 0,Y 277.274,Z 148.759,A -85,B 0,C 180,E1 -17490.481,E2 -17490.481} C_VEL
LIN {X 0,Y 277.249,Z 148.751,A -85,B 0,C 180,E1 -17493.896,E2 -17493.896} C_VEL
LIN {X 0,Y 277.269,Z 148.758,A -85,B 0,C 180,E1 -17497.469,E2 -17497.469} C_VEL
LIN {X 0,Y 277.211,Z 148.765,A -85,B 0,C 180,E1 -17501.236,E2 -17501.236} C_VEL
LIN {X 0,Y 277.203,Z 148.76,A -85,B 0,C 180,E1 -17505.226,E2 -17505.226} C_VEL
LIN {X 0,Y 277.224,Z 148.756,A -85,B 0,C 180,E1 -17509.512,E2 -17509.512} C_VEL
LIN {X 0,Y 277.283,Z 148.756,A -85,B 0,C 180,E1 -17512.533,E2 -17512.533} C_VEL
LIN {X 0,Y 277.25,Z 148.749,A -85,B 0,C 180,E1 -17516.104,E2 -17516.104} C_VEL
LIN {X 0,Y 277.263,Z 148.755,A -85,B 0,C 180,E1 -17519.538,E2 -17519.538} C_VEL
LIN {X 0,Y 277.377,Z 148.892,A -85,B 0,C 180,E1 -17523.855,E2 -17523.855} C_VEL
LIN {X 0,Y 278.888,Z 156.904,A -85,B 0,C 180,E1 -17527.193,E2 -17527.193} C_VEL
LIN {X 0,Y 279.873,Z 159.698,A -85,B 0,C 180,E1 -17527.429,E2 -17527.429} C_VEL
LIN {X 0,Y 282.778,Z 169.294,A -85,B 0,C 180,E1 -17527.933,E2 -17527.933} C_VEL
LIN {X 0,Y 286.039,Z 187.277,A -85,B 0,C 180,E1 -17528.676,E2 -17528.676} C_VEL
LIN {X 0,Y 285.013,Z 233.21,A -85,B 0,C 180,E1 -17529.852,E2 -17529.852} C_VEL
LIN {X 0,Y 284.544,Z 242.986,A -85,B 0,C 180,E1 -17530.287,E2 -17530.287} C_VEL
LIN {X 0,Y 283.781,Z 254.067,A -85,B 0,C 180,E1 -17531.031,E2 -17531.031} C_VEL
LIN {X 0,Y 282.635,Z 264.879,A -85,B 0,C 180,E1 -17532.078,E2 -17532.078} C_VEL
LIN {X 0,Y 281.605,Z 273.269,A -85,B 0,C 180,E1 -17533.134,E2 -17533.134} C_VEL
LIN {X 0,Y 280.532,Z 281.189,A -85,B 0,C 180,E1 -17534.376,E2 -17534.376} C_VEL
LIN {X 0,Y 279.718,Z 286.876,A -85,B 0,C 180,E1 -17535.448,E2 -17535.448} C_VEL
LIN {X 0,Y 278.666,Z 293.227,A -85,B 0,C 180,E1 -17536.88,E2 -17536.88} C_VEL
LIN {X 0,Y 277.587,Z 299.676,A -85,B 0,C 180,E1 -17538.684,E2 -17538.684} C_VEL
LIN {X 0,Y 276.788,Z 304.818,A -85,B 0,C 180,E1 -17540.5,E2 -17540.5} C_VEL
LIN {X 0,Y 276.086,Z 309.575,A -85,B 0,C 180,E1 -17542.687,E2 -17542.687} C_VEL
LIN {X 0,Y 275.766,Z 311.895,A -85,B 0,C 180,E1 -17544.149,E2 -17544.149} C_VEL
LIN {X 0,Y 275.548,Z 313.658,A -85,B 0,C 180,E1 -17545.611,E2 -17545.611} C_VEL
LIN {X 0,Y 275.377,Z 314.929,A -85,B 0,C 180,E1 -17547.074,E2 -17547.074} C_VEL
LIN {X 0,Y 275.26,Z 315.731,A -85,B 0,C 180,E1 -17548.537,E2 -17548.537} C_VEL
LIN {X 0,Y 275.234,Z 316.036,A -85,B 0,C 180,E1 -17550,E2 -17550} C_VEL
LIN {X 0,Y 275.26,Z 315.757,A -85,B 0,C 180,E1 -17551.463,E2 -17551.463} C_VEL
LIN {X 0,Y 275.375,Z 315.009,A -85,B 0,C 180,E1 -17552.925,E2 -17552.925} C_VEL
LIN {X 0,Y 275.542,Z 313.793,A -85,B 0,C 180,E1 -17554.388,E2 -17554.388} C_VEL
LIN {X 0,Y 275.821,Z 311.2,A -85,B 0,C 180,E1 -17556.418,E2 -17556.418} C_VEL
LIN {X 0,Y 276.27,Z 308.342,A -85,B 0,C 180,E1 -17558.042,E2 -17558.042} C_VEL
LIN {X 0,Y 277.027,Z 303.23,A -85,B 0,C 180,E1 -17560.229,E2 -17560.229} C_VEL
LIN {X 0,Y 277.981,Z 297.727,A -85,B 0,C 180,E1 -17562.039,E2 -17562.039} C_VEL
LIN {X 0,Y 279.09,Z 290.813,A -85,B 0,C 180,E1 -17563.841,E2 -17563.841} C_VEL
LIN {X 0,Y 280.308,Z 282.873,A -85,B 0,C 180,E1 -17565.449,E2 -17565.449} C_VEL
LIN {X 0,Y 281.359,Z 275.301,A -85,B 0,C 180,E1 -17566.693,E2 -17566.693} C_VEL
LIN {X 0,Y 282.453,Z 267.36,A -85,B 0,C 180,E1 -17567.746,E2 -17567.746} C_VEL
LIN {X 0,Y 283.386,Z 259.156,A -85,B 0,C 180,E1 -17568.62,E2 -17568.62} C_VEL
LIN {X 0,Y 284.123,Z 250.838,A -85,B 0,C 180,E1 -17569.319,E2 -17569.319} C_VEL
LIN {X 0,Y 284.735,Z 241.837,A -85,B 0,C 180,E1 -17569.886,E2 -17569.886} C_VEL
LIN {X 0,Y 285.136,Z 232.978,A -85,B 0,C 180,E1 -17570.27,E2 -17570.27} C_VEL
LIN {X 0,Y 286.04,Z 190.905,A -85,B 0,C 180,E1 -17571.351,E2 -17571.351} C_VEL
LIN {X 0,Y 285.883,Z 186.143,A -85,B 0,C 180,E1 -17571.489,E2 -17571.489} C_VEL
LIN {X 0,Y 282.414,Z 167.625,A -85,B 0,C 180,E1 -17572.266,E2 -17572.266} C_VEL
LIN {X 0,Y 279.018,Z 157.444,A -85,B 0,C 180,E1 -17572.849,E2 -17572.849} C_VEL
LIN {X 0,Y 278.75,Z 156.078,A -85,B 0,C 180,E1 -17573.193,E2 -17573.193} C_VEL
LIN {X 0,Y 277.373,Z 148.845,A -85,B 0,C 180,E1 -17576.321,E2 -17576.321} C_VEL
LIN {X 0,Y 277.272,Z 148.753,A -85,B 0,C 180,E1 -17580.481,E2 -17580.481} C_VEL
LIN {X 0,Y 277.254,Z 148.751,A -85,B 0,C 180,E1 -17583.894,E2 -17583.894} C_VEL
LIN {X 0,Y 277.281,Z 148.755,A -85,B 0,C 180,E1 -17587.467,E2 -17587.467} C_VEL
LIN {X 0,Y 277.209,Z 148.752,A -85,B 0,C 180,E1 -17591.236,E2 -17591.236} C_VEL
LIN {X 0,Y 277.2,Z 148.761,A -85,B 0,C 180,E1 -17595.226,E2 -17595.226} C_VEL
LIN {X 0,Y 277.222,Z 148.761,A -85,B 0,C 180,E1 -17599.512,E2 -17599.512} C_VEL
LIN {X 0,Y 277.267,Z 148.758,A -85,B 0,C 180,E1 -17602.53,E2 -17602.53} C_VEL
LIN {X 0,Y 277.246,Z 148.751,A -85,B 0,C 180,E1 -17606.104,E2 -17606.104} C_VEL
LIN {X 0,Y 277.26,Z 148.761,A -85,B 0,C 180,E1 -17609.538,E2 -17609.538} C_VEL
LIN {X 0,Y 277.356,Z 148.74,A -85,B 0,C 180,E1 -17612.864,E2 -17612.864} C_VEL
LIN {X 0,Y 277.327,Z 148.748,A -85,B 0,C 180,E1 -17616.079,E2 -17616.079} C_VEL
LIN {X 0,Y 277.344,Z 148.74,A -85,B 0,C 180,E1 -17620.766,E2 -17620.766} C_VEL
LIN {X 0,Y 277.434,Z 148.737,A -85,B 0,C 180,E1 -17625.326,E2 -17625.326} C_VEL
LIN {X 0,Y 277.451,Z 148.729,A -85,B 0,C 180,E1 -17629.113,E2 -17629.113} C_VEL
LIN {X 0,Y 276.817,Z 148.808,A -85,B 0,C 180,E1 -17630.326,E2 -17630.326} C_VEL
LIN {X 0,Y 273.924,Z 149.177,A -85,B 0,C 180,E1 -17632.301,E2 -17632.301} C_VEL
LIN {X 0,Y 271.477,Z 149.486,A -85,B 0,C 180,E1 -17633.906,E2 -17633.906} C_VEL
LIN {X 0,Y 270.477,Z 149.607,A -85,B 0,C 180,E1 -17635.152,E2 -17635.152} C_VEL
LIN {X 0,Y 270.425,Z 149.61,A -85,B 0,C 180,E1 -17635.574,E2 -17635.574} C_VEL
LIN {X 0,Y 270.786,Z 149.56,A -85,B 0,C 180,E1 -17638.513,E2 -17638.513} C_VEL
LIN {X 0,Y 270.786,Z 149.55,A -85,B 0,C 180,E1 -17641.487,E2 -17641.487} C_VEL
LIN {X 0,Y 270.611,Z 149.588,A -85,B 0,C 180,E1 -17647.461,E2 -17647.461} C_VEL
LIN {X 0,Y 270.44,Z 149.593,A -85,B 0,C 180,E1 -17650.481,E2 -17650.481} C_VEL
LIN {X 0,Y 270.401,Z 149.615,A -85,B 0,C 180,E1 -17655.065,E2 -17655.065} C_VEL
LIN {X 0,Y 270.3,Z 149.615,A -85,B 0,C 180,E1 -17659.755,E2 -17659.755} C_VEL
LIN {X 0,Y 270.273,Z 149.631,A -85,B 0,C 180,E1 -17664.586,E2 -17664.586} C_VEL
LIN {X 0,Y 270.271,Z 149.619,A -85,B 0,C 180,E1 -17667.909,E2 -17667.909} C_VEL
LIN {X 0,Y 270.183,Z 149.642,A -85,B 0,C 180,E1 -17671.348,E2 -17671.348} C_VEL
LIN {X 0,Y 270.2,Z 149.632,A -85,B 0,C 180,E1 -17674.906,E2 -17674.906} C_VEL
LIN {X 0,Y 270.196,Z 149.64,A -85,B 0,C 180,E1 -17678.711,E2 -17678.711} C_VEL
LIN {X 0,Y 270.169,Z 149.615,A -85,B 0,C 180,E1 -17682.559,E2 -17682.559} C_VEL
LIN {X 0,Y 270.163,Z 149.643,A -85,B 0,C 180,E1 -17686.751,E2 -17686.751} C_VEL
LIN {X 0,Y 270.172,Z 149.642,A -85,B 0,C 180,E1 -17689.434,E2 -17689.434} C_VEL
LIN {X 0,Y 270.239,Z 149.632,A -85,B 0,C 180,E1 -17693.727,E2 -17693.727} C_VEL
LIN {X 0,Y 270.202,Z 149.628,A -85,B 0,C 180,E1 -17696.893,E2 -17696.893} C_VEL
LIN {X 0,Y 270.272,Z 149.783,A -85,B 0,C 180,E1 -17699.994,E2 -17699.994} C_VEL
LIN {X 0,Y 272.019,Z 158.048,A -85,B 0,C 180,E1 -17703.534,E2 -17703.534} C_VEL
LIN {X 0,Y 273.107,Z 165.492,A -85,B 0,C 180,E1 -17706.492,E2 -17706.492} C_VEL
LIN {X 0,Y 273.133,Z 166.273,A -85,B 0,C 180,E1 -17706.645,E2 -17706.645} C_VEL
LIN {X 0,Y 277.665,Z 192.619,A -85,B 0,C 180,E1 -17707.806,E2 -17707.806} C_VEL
LIN {X 0,Y 279.177,Z 204.88,A -85,B 0,C 180,E1 -17708.264,E2 -17708.264} C_VEL
LIN {X 0,Y 278.257,Z 242.823,A -85,B 0,C 180,E1 -17709.263,E2 -17709.263} C_VEL
LIN {X 0,Y 277.644,Z 252.699,A -85,B 0,C 180,E1 -17709.706,E2 -17709.706} C_VEL
LIN {X 0,Y 276.625,Z 264.65,A -85,B 0,C 180,E1 -17710.534,E2 -17710.534} C_VEL
LIN {X 0,Y 275.632,Z 273.597,A -85,B 0,C 180,E1 -17711.415,E2 -17711.415} C_VEL
LIN {X 0,Y 274.53,Z 282.163,A -85,B 0,C 180,E1 -17712.495,E2 -17712.495} C_VEL
LIN {X 0,Y 273.248,Z 290.223,A -85,B 0,C 180,E1 -17713.758,E2 -17713.758} C_VEL
LIN {X 0,Y 272.194,Z 296.883,A -85,B 0,C 180,E1 -17715.037,E2 -17715.037} C_VEL
LIN {X 0,Y 271.158,Z 303.206,A -85,B 0,C 180,E1 -17716.511,E2 -17716.511} C_VEL
LIN {X 0,Y 270.283,Z 308.46,A -85,B 0,C 180,E1 -17717.994,E2 -17717.994} C_VEL
LIN {X 0,Y 269.603,Z 312.843,A -85,B 0,C 180,E1 -17719.486,E2 -17719.486} C_VEL
LIN {X 0,Y 268.832,Z 318.013,A -85,B 0,C 180,E1 -17721.733,E2 -17721.733} C_VEL
LIN {X 0,Y 268.347,Z 321.808,A -85,B 0,C 180,E1 -17723.987,E2 -17723.987} C_VEL
LIN {X 0,Y 268.206,Z 323.552,A -85,B 0,C 180,E1 -17725.492,E2 -17725.492} C_VEL
LIN {X 0,Y 268.171,Z 324.801,A -85,B 0,C 180,E1 -17726.996,E2 -17726.996} C_VEL
LIN {X 0,Y 268.137,Z 325.575,A -85,B 0,C 180,E1 -17728.498,E2 -17728.498} C_VEL
LIN {X 0,Y 268.154,Z 325.868,A -85,B 0,C 180,E1 -17730,E2 -17730} C_VEL
LIN {X 0,Y 268.137,Z 325.568,A -85,B 0,C 180,E1 -17731.502,E2 -17731.502} C_VEL
LIN {X 0,Y 268.171,Z 324.779,A -85,B 0,C 180,E1 -17733.005,E2 -17733.005} C_VEL
LIN {X 0,Y 268.308,Z 322.421,A -85,B 0,C 180,E1 -17735.521,E2 -17735.521} C_VEL
LIN {X 0,Y 268.637,Z 319.427,A -85,B 0,C 180,E1 -17737.517,E2 -17737.517} C_VEL
LIN {X 0,Y 269.254,Z 314.673,A -85,B 0,C 180,E1 -17739.768,E2 -17739.768} C_VEL
LIN {X 0,Y 270.094,Z 309.527,A -85,B 0,C 180,E1 -17741.634,E2 -17741.634} C_VEL
LIN {X 0,Y 270.941,Z 304.497,A -85,B 0,C 180,E1 -17743.119,E2 -17743.119} C_VEL
LIN {X 0,Y 271.904,Z 298.439,A -85,B 0,C 180,E1 -17744.597,E2 -17744.597} C_VEL
LIN {X 0,Y 273.121,Z 291.069,A -85,B 0,C 180,E1 -17746.059,E2 -17746.059} C_VEL
LIN {X 0,Y 274.324,Z 283.175,A -85,B 0,C 180,E1 -17747.327,E2 -17747.327} C_VEL
LIN {X 0,Y 275.449,Z 274.829,A -85,B 0,C 180,E1 -17748.406,E2 -17748.406} C_VEL
LIN {X 0,Y 276.592,Z 264.28,A -85,B 0,C 180,E1 -17749.47,E2 -17749.47} C_VEL
LIN {X 0,Y 277.598,Z 252.82,A -85,B 0,C 180,E1 -17750.257,E2 -17750.257} C_VEL
LIN {X 0,Y 278.209,Z 243.86,A -85,B 0,C 180,E1 -17750.668,E2 -17750.668} C_VEL
LIN {X 0,Y 278.908,Z 212.828,A -85,B 0,C 180,E1 -17751.508,E2 -17751.508} C_VEL
LIN {X 0,Y 278.901,Z 201.82,A -85,B 0,C 180,E1 -17751.806,E2 -17751.806} C_VEL
LIN {X 0,Y 275.149,Z 177.417,A -85,B 0,C 180,E1 -17752.791,E2 -17752.791} C_VEL
LIN {X 0,Y 273.044,Z 166.083,A -85,B 0,C 180,E1 -17753.341,E2 -17753.341} C_VEL
LIN {X 0,Y 272.881,Z 163.202,A -85,B 0,C 180,E1 -17754.336,E2 -17754.336} C_VEL
LIN {X 0,Y 271.379,Z 154.791,A -85,B 0,C 180,E1 -17757.785,E2 -17757.785} C_VEL
LIN {X 0,Y 270.274,Z 149.714,A -85,B 0,C 180,E1 -17760.007,E2 -17760.007} C_VEL
LIN {X 0,Y 270.217,Z 149.627,A -85,B 0,C 180,E1 -17763.667,E2 -17763.667} C_VEL
LIN {X 0,Y 270.226,Z 149.63,A -85,B 0,C 180,E1 -17766.74,E2 -17766.74} C_VEL
LIN {X 0,Y 270.17,Z 149.642,A -85,B 0,C 180,E1 -17771.029,E2 -17771.029} C_VEL
LIN {X 0,Y 270.152,Z 149.621,A -85,B 0,C 180,E1 -17775.38,E2 -17775.38} C_VEL
LIN {X 0,Y 270.174,Z 149.634,A -85,B 0,C 180,E1 -17779.434,E2 -17779.434} C_VEL
LIN {X 0,Y 270.227,Z 149.632,A -85,B 0,C 180,E1 -17783.731,E2 -17783.731} C_VEL
LIN {X 0,Y 270.204,Z 149.636,A -85,B 0,C 180,E1 -17786.893,E2 -17786.893} C_VEL
LIN {X 0,Y 270.231,Z 149.633,A -85,B 0,C 180,E1 -17790.387,E2 -17790.387} C_VEL
LIN {X 0,Y 270.267,Z 149.627,A -85,B 0,C 180,E1 -17793.764,E2 -17793.764} C_VEL
LIN {X 0,Y 270.235,Z 149.635,A -85,B 0,C 180,E1 -17797.039,E2 -17797.039} C_VEL
LIN {X 0,Y 270.303,Z 149.614,A -85,B 0,C 180,E1 -17800.245,E2 -17800.245} C_VEL
LIN {X 0,Y 270.405,Z 149.615,A -85,B 0,C 180,E1 -17804.936,E2 -17804.936} C_VEL
LIN {X 0,Y 270.415,Z 149.595,A -85,B 0,C 180,E1 -17809.518,E2 -17809.518} C_VEL
LIN {X 0,Y 270.6,Z 149.589,A -85,B 0,C 180,E1 -17812.539,E2 -17812.539} C_VEL
LIN {X 0,Y 270.788,Z 149.55,A -85,B 0,C 180,E1 -17818.513,E2 -17818.513} C_VEL
LIN {X 0,Y 270.788,Z 149.559,A -85,B 0,C 180,E1 -17821.487,E2 -17821.487} C_VEL
LIN {X 0,Y 270.613,Z 149.58,A -85,B 0,C 180,E1 -17827.461,E2 -17827.461} C_VEL
LIN {X 0,Y 270.444,Z 149.601,A -85,B 0,C 180,E1 -17830.481,E2 -17830.481} C_VEL
LIN {X 0,Y 270.405,Z 149.614,A -85,B 0,C 180,E1 -17835.065,E2 -17835.065} C_VEL
LIN {X 0,Y 270.304,Z 149.621,A -85,B 0,C 180,E1 -17839.756,E2 -17839.756} C_VEL
LIN {X 0,Y 270.276,Z 149.627,A -85,B 0,C 180,E1 -17844.586,E2 -17844.586} C_VEL
LIN {X 0,Y 270.274,Z 149.624,A -85,B 0,C 180,E1 -17847.909,E2 -17847.909} C_VEL
LIN {X 0,Y 270.186,Z 149.64,A -85,B 0,C 180,E1 -17851.348,E2 -17851.348} C_VEL
LIN {X 0,Y 270.204,Z 149.634,A -85,B 0,C 180,E1 -17854.905,E2 -17854.905} C_VEL
LIN {X 0,Y 270.199,Z 149.637,A -85,B 0,C 180,E1 -17858.71,E2 -17858.71} C_VEL
LIN {X 0,Y 270.167,Z 149.644,A -85,B 0,C 180,E1 -17863.249,E2 -17863.249} C_VEL
LIN {X 0,Y 270.173,Z 149.618,A -85,B 0,C 180,E1 -17867.442,E2 -17867.442} C_VEL
LIN {X 0,Y 270.209,Z 149.638,A -85,B 0,C 180,E1 -17871.374,E2 -17871.374} C_VEL
LIN {X 0,Y 270.213,Z 149.619,A -85,B 0,C 180,E1 -17875.096,E2 -17875.096} C_VEL
LIN {X 0,Y 270.202,Z 149.637,A -85,B 0,C 180,E1 -17879.13,E2 -17879.13} C_VEL
LIN {X 0,Y 270.326,Z 149.805,A -85,B 0,C 180,E1 -17883.458,E2 -17883.458} C_VEL
LIN {X 0,Y 271.669,Z 156.834,A -85,B 0,C 180,E1 -17886.511,E2 -17886.511} C_VEL
LIN {X 0,Y 272.142,Z 158.483,A -85,B 0,C 180,E1 -17886.711,E2 -17886.711} C_VEL
LIN {X 0,Y 275.849,Z 168.95,A -85,B 0,C 180,E1 -17887.335,E2 -17887.335} C_VEL
LIN {X 0,Y 279.424,Z 188.179,A -85,B 0,C 180,E1 -17888.166,E2 -17888.166} C_VEL
LIN {X 0,Y 278.376,Z 233.355,A -85,B 0,C 180,E1 -17889.35,E2 -17889.35} C_VEL
LIN {X 0,Y 277.885,Z 243.125,A -85,B 0,C 180,E1 -17889.795,E2 -17889.795} C_VEL
LIN {X 0,Y 277.1,Z 254.203,A -85,B 0,C 180,E1 -17890.556,E2 -17890.556} C_VEL
LIN {X 0,Y 275.897,Z 265.013,A -85,B 0,C 180,E1 -17891.625,E2 -17891.625} C_VEL
LIN {X 0,Y 274.844,Z 273.401,A -85,B 0,C 180,E1 -17892.707,E2 -17892.707} C_VEL
LIN {X 0,Y 273.709,Z 281.321,A -85,B 0,C 180,E1 -17893.976,E2 -17893.976} C_VEL
LIN {X 0,Y 272.842,Z 287.007,A -85,B 0,C 180,E1 -17895.073,E2 -17895.073} C_VEL
LIN {X 0,Y 271.746,Z 293.358,A -85,B 0,C 180,E1 -17896.54,E2 -17896.54} C_VEL
LIN {X 0,Y 270.618,Z 299.806,A -85,B 0,C 180,E1 -17898.388,E2 -17898.388} C_VEL
LIN {X 0,Y 269.797,Z 304.948,A -85,B 0,C 180,E1 -17900.251,E2 -17900.251} C_VEL
LIN {X 0,Y 269.045,Z 309.705,A -85,B 0,C 180,E1 -17902.495,E2 -17902.495} C_VEL
LIN {X 0,Y 268.717,Z 312.024,A -85,B 0,C 180,E1 -17903.995,E2 -17903.995} C_VEL
LIN {X 0,Y 268.462,Z 313.787,A -85,B 0,C 180,E1 -17905.495,E2 -17905.495} C_VEL
LIN {X 0,Y 268.294,Z 315.058,A -85,B 0,C 180,E1 -17906.997,E2 -17906.997} C_VEL
LIN {X 0,Y 268.19,Z 315.859,A -85,B 0,C 180,E1 -17908.498,E2 -17908.498} C_VEL
LIN {X 0,Y 268.16,Z 316.164,A -85,B 0,C 180,E1 -17910,E2 -17910} C_VEL
LIN {X 0,Y 268.19,Z 315.885,A -85,B 0,C 180,E1 -17911.501,E2 -17911.501} C_VEL
LIN {X 0,Y 268.292,Z 315.137,A -85,B 0,C 180,E1 -17913.003,E2 -17913.003} C_VEL
LIN {X 0,Y 268.454,Z 313.921,A -85,B 0,C 180,E1 -17914.504,E2 -17914.504} C_VEL
LIN {X 0,Y 268.71,Z 311.699,A -85,B 0,C 180,E1 -17916.344,E2 -17916.344} C_VEL
LIN {X 0,Y 269.235,Z 308.469,A -85,B 0,C 180,E1 -17918.254,E2 -17918.254} C_VEL
LIN {X 0,Y 270.034,Z 303.357,A -85,B 0,C 180,E1 -17920.497,E2 -17920.497} C_VEL
LIN {X 0,Y 271.022,Z 297.854,A -85,B 0,C 180,E1 -17922.353,E2 -17922.353} C_VEL
LIN {X 0,Y 272.207,Z 290.939,A -85,B 0,C 180,E1 -17924.198,E2 -17924.198} C_VEL
LIN {X 0,Y 273.468,Z 282.998,A -85,B 0,C 180,E1 -17925.846,E2 -17925.846} C_VEL
LIN {X 0,Y 274.582,Z 275.425,A -85,B 0,C 180,E1 -17927.118,E2 -17927.118} C_VEL
LIN {X 0,Y 275.713,Z 267.483,A -85,B 0,C 180,E1 -17928.195,E2 -17928.195} C_VEL
LIN {X 0,Y 276.678,Z 259.278,A -85,B 0,C 180,E1 -17929.089,E2 -17929.089} C_VEL
LIN {X 0,Y 277.456,Z 250.958,A -85,B 0,C 180,E1 -17929.803,E2 -17929.803} C_VEL
LIN {X 0,Y 278.093,Z 241.954,A -85,B 0,C 180,E1 -17930.382,E2 -17930.382} C_VEL
LIN {X 0,Y 278.505,Z 232.967,A -85,B 0,C 180,E1 -17930.779,E2 -17930.779} C_VEL
LIN {X 0,Y 279.441,Z 191.009,A -85,B 0,C 180,E1 -17931.881,E2 -17931.881} C_VEL
LIN {X 0,Y 279.284,Z 187.185,A -85,B 0,C 180,E1 -17931.998,E2 -17931.998} C_VEL
LIN {X 0,Y 276.034,Z 169.655,A -85,B 0,C 180,E1 -17932.756,E2 -17932.756} C_VEL
LIN {X 0,Y 272.46,Z 159.272,A -85,B 0,C 180,E1 -17933.365,E2 -17933.365} C_VEL
LIN {X 0,Y 271.711,Z 156.988,A -85,B 0,C 180,E1 -17933.585,E2 -17933.585} C_VEL
LIN {X 0,Y 270.352,Z 149.774,A -85,B 0,C 180,E1 -17936.694,E2 -17936.694} C_VEL
LIN {X 0,Y 270.185,Z 149.64,A -85,B 0,C 180,E1 -17941.348,E2 -17941.348} C_VEL
LIN {X 0,Y 270.215,Z 149.619,A -85,B 0,C 180,E1 -17944.903,E2 -17944.903} C_VEL
LIN {X 0,Y 270.222,Z 149.637,A -85,B 0,C 180,E1 -17948.717,E2 -17948.717} C_VEL
LIN {X 0,Y 270.164,Z 149.618,A -85,B 0,C 180,E1 -17953.248,E2 -17953.248} C_VEL
LIN {X 0,Y 270.171,Z 149.646,A -85,B 0,C 180,E1 -17957.441,E2 -17957.441} C_VEL
LIN {X 0,Y 270.206,Z 149.636,A -85,B 0,C 180,E1 -17961.374,E2 -17961.374} C_VEL
LIN {X 0,Y 270.201,Z 149.635,A -85,B 0,C 180,E1 -17965.094,E2 -17965.094} C_VEL
LIN {X 0,Y 270.199,Z 149.641,A -85,B 0,C 180,E1 -17969.13,E2 -17969.13} C_VEL
